C09156=1163.413,-13.561,-45.974,179.721,5.975,149.153
C09157=1163.408,-13.312,-45.986,179.723,5.976,149.152
C09158=1163.403,-13.062,-45.999,179.726,5.976,149.151
C09159=1163.397,-12.812,-46.012,179.728,5.977,149.151
C09160=1163.392,-12.563,-46.025,179.731,5.978,149.150
C09161=1163.388,-12.313,-46.038,179.733,5.978,149.150
C09162=1163.383,-12.063,-46.050,179.736,5.979,149.149
C09163=1163.377,-11.814,-46.064,179.738,5.979,149.148
C09164=1163.372,-11.564,-46.077,179.740,5.980,149.148
C09165=1163.367,-11.314,-46.089,179.743,5.981,149.147
C09166=1163.361,-11.065,-46.102,179.745,5.981,149.147
C09167=1163.356,-10.815,-46.115,179.748,5.982,149.146
C09168=1163.352,-10.565,-46.128,179.750,5.983,149.146
C09169=1163.346,-10.316,-46.141,179.753,5.983,149.145
C09170=1163.341,-10.066,-46.154,179.755,5.984,149.144
C09171=1163.336,-9.816,-46.167,179.758,5.984,149.144
C09172=1163.330,-9.567,-46.180,179.760,5.985,149.143
C09173=1163.326,-9.317,-46.193,179.763,5.986,149.143
C09174=1163.321,-9.067,-46.206,179.766,5.987,149.142
C09175=1163.315,-8.818,-46.219,179.768,5.988,149.141
C09176=1163.311,-8.568,-46.232,179.770,5.988,149.141
C09177=1163.305,-8.319,-46.245,179.773,5.989,149.140
C09178=1163.300,-8.069,-46.258,179.775,5.989,149.140
C09179=1163.295,-7.819,-46.271,179.778,5.990,149.139
C09180=1163.290,-7.570,-46.284,179.780,5.991,149.138
C09181=1163.284,-7.321,-46.297,179.783,5.991,149.138
C09182=1163.280,-7.071,-46.311,179.785,5.992,149.137
C09183=1163.274,-6.822,-46.324,179.788,5.992,149.137
C09184=1163.269,-6.571,-46.337,179.790,5.993,149.136
C09185=1163.264,-6.322,-46.349,179.792,5.994,149.135
C09186=1163.258,-6.073,-46.363,179.795,5.994,149.135
C09187=1163.254,-5.823,-46.376,179.797,5.995,149.134
C09188=1163.248,-5.574,-46.389,179.800,5.995,149.134
C09189=1163.244,-5.323,-46.402,179.802,5.996,149.133
C09190=1163.238,-5.074,-46.416,179.805,5.997,149.132
C09191=1163.233,-4.825,-46.429,179.807,5.997,149.132
C09192=1163.229,-4.575,-46.442,179.810,5.998,149.131
C09193=1163.223,-4.326,-46.455,179.812,5.998,149.131
C09194=1163.218,-4.075,-46.468,179.814,5.999,149.130
C09195=1163.213,-3.826,-46.482,179.817,6.000,149.129
C09196=1163.208,-3.576,-46.495,179.819,6.000,149.129
C09197=1163.202,-3.327,-46.508,179.822,6.002,149.128
C09198=1163.198,-3.077,-46.521,179.825,6.002,149.128
C09199=1163.192,-2.828,-46.535,179.827,6.003,149.127
C09200=1163.187,-2.578,-46.548,179.830,6.003,149.126
C09201=1163.182,-2.328,-46.561,179.832,6.004,149.126
C09202=1163.177,-2.079,-46.575,179.835,6.005,149.125
C09203=1163.172,-1.829,-46.588,179.837,6.006,149.125
C09204=1163.167,-1.580,-46.601,179.840,6.006,149.124
C09205=1163.162,-1.330,-46.615,179.842,6.007,149.124
C09206=1163.157,-1.081,-46.628,179.844,6.007,149.123
C09207=1163.152,-0.831,-46.642,179.847,6.008,149.122
C09208=1163.146,-0.581,-46.655,179.849,6.009,149.122
C09209=1163.141,-0.331,-46.668,179.852,6.009,149.121
C09210=1163.136,-0.082,-46.682,179.854,6.010,149.121
C09211=1163.131,0.168,-46.695,179.857,6.010,149.120
C09212=1163.126,0.417,-46.709,179.860,6.012,149.120
C09213=1163.121,0.667,-46.722,179.862,6.012,149.119
C09214=1163.115,0.916,-46.735,179.865,6.013,149.118
C09215=1163.110,1.166,-46.749,179.867,6.014,149.118
C09216=1163.105,1.415,-46.762,179.870,6.014,149.117
C09217=1163.100,1.685,-46.777,179.872,6.015,149.117
C09218=1163.094,1.954,-46.792,179.874,6.015,149.116
C09219=1163.088,2.223,-46.806,179.878,6.017,149.115
C09220=1163.083,2.493,-46.820,179.880,6.017,149.114
C09221=1163.078,2.742,-46.834,179.883,6.018,149.114
C09222=1163.072,2.992,-46.848,179.885,6.018,149.113
C09223=1163.068,3.241,-46.861,179.887,6.019,149.113
C09224=1163.062,3.491,-46.874,179.890,6.020,149.112
C09225=1163.057,3.741,-46.889,179.893,6.020,149.111
C09226=1163.052,3.990,-46.901,179.895,6.021,149.111
C09227=1163.047,4.240,-46.916,179.898,6.022,149.110
C09228=1163.043,4.490,-46.929,179.900,6.023,149.110
C09229=1163.037,4.739,-46.942,179.903,6.023,149.109
C09230=1163.032,4.988,-46.957,179.905,6.024,149.109
C09231=1163.026,5.238,-46.970,179.908,6.025,149.108
C09232=1163.022,5.487,-46.984,179.910,6.026,149.108
C09233=1163.016,5.737,-46.997,179.913,6.026,149.107
C09234=1163.011,5.987,-47.011,179.915,6.027,149.106
C09235=1163.007,6.236,-47.025,179.917,6.027,149.106
C09236=1163.001,6.486,-47.038,179.921,6.029,149.105
C09237=1162.996,6.736,-47.052,179.923,6.029,149.105
C09238=1162.991,6.985,-47.065,179.925,6.030,149.104
C09239=1162.986,7.235,-47.079,179.928,6.031,149.103
C09240=1162.981,7.484,-47.093,179.930,6.031,149.103
C09241=1162.975,7.734,-47.107,179.933,6.032,149.102
C09242=1162.971,7.983,-47.120,179.935,6.032,149.102
C09243=1162.966,8.233,-47.135,179.938,6.033,149.101
C09244=1162.961,8.482,-47.149,179.941,6.035,149.100
C09245=1162.955,8.732,-47.162,179.943,6.035,149.100
C09246=1162.950,8.981,-47.176,179.945,6.036,149.099
C09247=1162.946,9.231,-47.190,179.948,6.036,149.099
C09248=1162.940,9.481,-47.203,179.950,6.037,149.098
C09249=1162.935,9.730,-47.217,179.953,6.038,149.097
C09250=1162.930,9.980,-47.231,179.955,6.038,149.097
C09251=1162.925,10.229,-47.246,179.958,6.039,149.096
C09252=1162.920,10.479,-47.258,179.961,6.040,149.096
C09253=1162.915,10.729,-47.273,179.963,6.041,149.095
C09254=1162.910,10.978,-47.287,179.966,6.041,149.095
C09255=1162.904,11.227,-47.301,179.968,6.042,149.094
C09256=1162.899,11.478,-47.314,179.971,6.043,149.093
C09257=1162.894,11.727,-47.329,179.973,6.044,149.093
C09258=1162.889,11.976,-47.342,179.975,6.044,149.092
C09259=1162.884,12.226,-47.356,179.979,6.045,149.092
C09260=1162.879,12.475,-47.370,179.981,6.046,149.091
C09261=1162.874,12.724,-47.384,179.983,6.047,149.090
C09262=1162.869,12.975,-47.398,179.986,6.047,149.090
C09263=1162.864,13.224,-47.412,179.988,6.048,149.089
C09264=1162.859,13.474,-47.426,179.990,6.049,149.089
C09265=1162.854,13.723,-47.440,179.993,6.049,149.088
C09266=1162.849,13.973,-47.454,179.996,6.051,149.088
C09267=1162.844,14.222,-47.468,179.998,6.051,149.087
C09268=1162.838,14.471,-47.482,-179.999,6.052,149.086
C09269=1162.833,14.721,-47.497,-179.997,6.053,149.086
C09270=1162.829,14.971,-47.511,-179.994,6.053,149.085
C09271=1162.823,15.221,-47.524,-179.992,6.054,149.085
C09272=1162.818,15.470,-47.538,-179.989,6.055,149.084
C09273=1162.813,15.720,-47.553,-179.986,6.056,149.084
C09274=1162.808,15.969,-47.567,-179.984,6.056,149.083
C09275=1162.803,16.219,-47.581,-179.982,6.057,149.082
C09276=1162.797,16.468,-47.595,-179.979,6.058,149.082
C09277=1162.792,16.718,-47.609,-179.977,6.059,149.081
C09278=1162.787,16.968,-47.624,-179.974,6.060,149.081
C09279=1162.782,17.217,-47.638,-179.971,6.060,149.080
C09280=1162.777,17.466,-47.652,-179.969,6.061,149.079
C09281=1162.772,17.716,-47.666,-179.966,6.062,149.079
C09282=1162.767,17.966,-47.680,-179.964,6.062,149.078
C09283=1162.762,18.215,-47.695,-179.961,6.064,149.078
C09284=1162.757,18.465,-47.709,-179.959,6.065,149.077
C09285=1162.751,18.714,-47.723,-179.956,6.065,149.076
C09286=1162.747,18.964,-47.737,-179.954,6.066,149.076
C09287=1162.742,19.214,-47.751,-179.951,6.066,149.075
C09288=1162.737,19.463,-47.766,-179.948,6.068,149.075
C09289=1162.732,19.712,-47.781,-179.946,6.068,149.074
C09290=1162.726,19.961,-47.795,-179.943,6.069,149.074
C09291=1162.721,20.211,-47.809,-179.941,6.070,149.073
C09292=1162.717,20.461,-47.823,-179.938,6.070,149.072
C09293=1162.712,20.711,-47.837,-179.936,6.071,149.072
C09294=1162.707,20.960,-47.852,-179.933,6.072,149.071
C09295=1162.702,21.210,-47.866,-179.931,6.073,149.071
C09296=1162.696,21.459,-47.880,-179.928,6.074,149.070
C09297=1162.691,21.708,-47.895,-179.926,6.074,149.070
C09298=1162.686,21.958,-47.909,-179.923,6.076,149.069
C09299=1162.682,22.207,-47.923,-179.920,6.077,149.069
C09300=1162.676,22.458,-47.938,-179.918,6.077,149.068
C09301=1162.671,22.707,-47.953,-179.915,6.078,149.067
C09302=1162.666,22.956,-47.968,-179.913,6.078,149.067
C09303=1162.661,23.205,-47.981,-179.910,6.080,149.066
C09304=1162.656,23.455,-47.996,-179.908,6.080,149.066
C09305=1162.651,23.705,-48.010,-179.905,6.081,149.065
C09306=1162.646,23.954,-48.024,-179.903,6.082,149.064
C09307=1162.640,24.204,-48.040,-179.900,6.082,149.064
C09308=1162.635,24.454,-48.054,-179.897,6.084,149.063
C09309=1162.631,24.703,-48.068,-179.895,6.084,149.063
C09310=1162.626,24.953,-48.083,-179.893,6.085,149.062
C09311=1162.621,25.202,-48.098,-179.890,6.086,149.062
C09312=1162.615,25.451,-48.112,-179.887,6.087,149.061
C09313=1162.610,25.701,-48.126,-179.884,6.088,149.060
C09314=1162.605,25.950,-48.141,-179.882,6.088,149.060
C09315=1162.600,26.200,-48.156,-179.880,6.089,149.059
C09316=1162.595,26.450,-48.170,-179.877,6.090,149.059
C09317=1162.590,26.699,-48.185,-179.874,6.091,149.058
C09318=1162.585,26.949,-48.200,-179.872,6.092,149.057
C09319=1162.580,27.198,-48.214,-179.869,6.093,149.057
C09320=1162.575,27.448,-48.229,-179.867,6.093,149.056
C09321=1162.570,27.717,-48.244,-179.864,6.095,149.056
C09322=1162.564,27.986,-48.260,-179.861,6.095,149.055
C09323=1162.559,28.255,-48.276,-179.858,6.096,149.054
C09324=1162.554,28.524,-48.292,-179.856,6.097,149.054
C09325=1162.548,28.772,-48.307,-179.853,6.098,149.053
C09326=1162.543,29.022,-48.321,-179.850,6.099,149.053
C09327=1162.538,29.272,-48.336,-179.848,6.100,149.052
C09328=1162.532,29.521,-48.351,-179.845,6.100,149.052
C09329=1162.527,29.771,-48.365,-179.843,6.101,149.051
C09330=1162.523,30.020,-48.380,-179.840,6.102,149.050
C09331=1162.518,30.270,-48.395,-179.838,6.103,149.050
C09332=1162.512,30.519,-48.410,-179.835,6.104,149.049
C09333=1162.507,30.769,-48.425,-179.833,6.105,149.049
C09334=1162.503,31.018,-48.440,-179.830,6.106,149.048
C09335=1162.497,31.268,-48.454,-179.828,6.107,149.048
C09336=1162.492,31.517,-48.469,-179.825,6.107,149.047
C09337=1162.487,31.767,-48.484,-179.823,6.108,149.047
C09338=1162.482,32.016,-48.499,-179.820,6.109,149.046
C09339=1162.477,32.266,-48.514,-179.817,6.110,149.045
C09340=1162.472,32.515,-48.529,-179.815,6.111,149.045
C09341=1162.467,32.765,-48.543,-179.811,6.112,149.044
C09342=1162.462,33.014,-48.558,-179.809,6.113,149.044
C09343=1162.458,33.264,-48.573,-179.807,6.113,149.043
C09344=1162.452,33.514,-48.589,-179.805,6.114,149.043
C09345=1162.448,33.763,-48.604,-179.801,6.115,149.042
C09346=1162.442,34.013,-48.619,-179.799,6.116,149.041
C09347=1162.437,34.262,-48.634,-179.796,6.117,149.041
C09348=1162.432,34.512,-48.648,-179.794,6.118,149.040
C09349=1162.427,34.761,-48.663,-179.791,6.119,149.040
C09350=1162.422,35.010,-48.678,-179.789,6.120,149.039
C09351=1162.417,35.260,-48.693,-179.786,6.120,149.038
C09352=1162.412,35.509,-48.708,-179.784,6.122,149.038
C09353=1162.407,35.759,-48.724,-179.781,6.122,149.037
C09354=1162.402,36.008,-48.738,-179.779,6.123,149.037
C09355=1162.396,36.258,-48.754,-179.775,6.124,149.036
C09356=1162.392,36.507,-48.769,-179.773,6.125,149.036
C09357=1162.386,36.757,-48.784,-179.771,6.126,149.035
C09358=1162.382,37.007,-48.799,-179.769,6.127,149.035
C09359=1162.377,37.256,-48.814,-179.765,6.128,149.034
C09360=1162.372,37.506,-48.829,-179.763,6.129,149.034
C09361=1162.367,37.755,-48.844,-179.760,6.129,149.033
C09362=1162.362,38.004,-48.859,-179.758,6.131,149.032
C09363=1162.357,38.253,-48.874,-179.755,6.131,149.032
C09364=1162.351,38.503,-48.889,-179.753,6.132,149.031
C09365=1162.346,38.753,-48.905,-179.750,6.134,149.031
C09366=1162.341,39.002,-48.920,-179.748,6.134,149.030
C09367=1162.336,39.252,-48.936,-179.745,6.135,149.030
C09368=1162.331,39.502,-48.950,-179.742,6.137,149.029
C09369=1162.326,39.751,-48.966,-179.739,6.137,149.028
C09370=1162.321,40.000,-48.981,-179.737,6.138,149.028
C09371=1162.316,40.250,-48.996,-179.735,6.138,149.027
C09372=1162.311,40.499,-49.011,-179.732,6.140,149.027
C09373=1162.306,40.748,-49.027,-179.729,6.140,149.026
C09374=1162.301,40.999,-49.042,-179.727,6.141,149.026
C09375=1162.296,41.248,-49.057,-179.724,6.143,149.025
C09376=1162.291,41.497,-49.073,-179.722,6.143,149.025
C09377=1162.286,41.746,-49.088,-179.719,6.144,149.024
C09378=1162.281,41.996,-49.103,-179.716,6.146,149.023
C09379=1162.277,42.246,-49.119,-179.714,6.146,149.023
C09380=1162.271,42.495,-49.134,-179.712,6.147,149.022
C09381=1162.266,42.744,-49.150,-179.708,6.148,149.022
C09382=1162.261,42.994,-49.165,-179.706,6.149,149.021
C09383=1162.256,43.244,-49.180,-179.704,6.150,149.021
C09384=1162.251,43.494,-49.196,-179.701,6.151,149.020
C09385=1162.246,43.743,-49.211,-179.698,6.152,149.019
C09386=1162.241,43.992,-49.226,-179.696,6.153,149.019
C09387=1162.235,44.242,-49.242,-179.693,6.154,149.018
C09388=1162.231,44.491,-49.257,-179.691,6.155,149.018
C09389=1162.226,44.741,-49.273,-179.687,6.156,149.017
C09390=1162.221,44.990,-49.288,-179.685,6.157,149.017
C09391=1162.216,45.239,-49.303,-179.683,6.157,149.016
C09392=1162.211,45.489,-49.319,-179.680,6.159,149.016
C09393=1162.206,45.739,-49.335,-179.677,6.160,149.015
C09394=1162.201,45.988,-49.350,-179.675,6.160,149.015
C09395=1162.196,46.237,-49.365,-179.672,6.162,149.014
C09396=1162.190,46.487,-49.381,-179.670,6.163,149.013
C09397=1162.186,46.737,-49.397,-179.667,6.163,149.013
C09398=1162.181,46.985,-49.413,-179.664,6.165,149.012
C09399=1162.176,47.235,-49.428,-179.662,6.165,149.012
C09400=1162.171,47.484,-49.444,-179.659,6.166,149.011
C09401=1162.166,47.734,-49.459,-179.656,6.167,149.011
C09402=1162.161,47.983,-49.475,-179.654,6.168,149.010
C09403=1162.156,48.233,-49.490,-179.651,6.169,149.009
C09404=1162.151,48.483,-49.506,-179.649,6.170,149.009
C09405=1162.146,48.732,-49.522,-179.646,6.171,149.008
C09406=1162.141,48.981,-49.537,-179.643,6.172,149.008
C09407=1162.136,49.231,-49.554,-179.641,6.173,149.007
C09408=1162.131,49.480,-49.569,-179.638,6.174,149.007
C09409=1162.126,49.730,-49.585,-179.635,6.175,149.006
C09410=1162.121,49.979,-49.600,-179.633,6.176,149.006
C09411=1162.116,50.229,-49.616,-179.630,6.178,149.005
C09412=1162.111,50.478,-49.632,-179.628,6.178,149.005
C09413=1162.106,50.727,-49.648,-179.626,6.179,149.004
C09414=1162.101,50.977,-49.664,-179.622,6.180,149.003
C09415=1162.096,51.226,-49.679,-179.620,6.181,149.003
C09416=1162.091,51.476,-49.694,-179.617,6.182,149.002
C09417=1162.086,51.725,-49.711,-179.615,6.183,149.002
C09418=1162.081,51.974,-49.726,-179.612,6.184,149.001
C09419=1162.076,52.225,-49.742,-179.609,6.185,149.001
C09420=1162.071,52.474,-49.758,-179.607,6.186,149.000
C09421=1162.066,52.723,-49.774,-179.604,6.188,149.000
C09422=1162.061,52.973,-49.790,-179.601,6.188,148.999
C09423=1162.056,53.222,-49.806,-179.599,6.189,148.999
C09424=1162.051,53.471,-49.821,-179.596,6.190,148.998
C09425=1162.046,53.740,-49.839,-179.594,6.191,148.997
C09426=1162.041,54.008,-49.856,-179.591,6.192,148.997
C09427=1162.035,54.277,-49.873,-179.587,6.194,148.996
C09428=1162.030,54.545,-49.890,-179.585,6.195,148.996
C09429=1162.025,54.795,-49.906,-179.582,6.196,148.995
C09430=1162.020,55.044,-49.922,-179.580,6.197,148.995
C09431=1162.015,55.294,-49.938,-179.577,6.197,148.994
C09432=1162.010,55.544,-49.954,-179.574,6.199,148.993
C09433=1162.005,55.792,-49.970,-179.572,6.199,148.993
C09434=1162.000,56.043,-49.986,-179.569,6.201,148.992
C09435=1161.995,56.291,-50.002,-179.567,6.202,148.992
C09436=1161.990,56.541,-50.018,-179.564,6.203,148.991
C09437=1161.985,56.790,-50.035,-179.562,6.204,148.991
C09438=1161.980,57.040,-50.050,-179.559,6.205,148.990
C09439=1161.975,57.290,-50.066,-179.556,6.206,148.990
C09440=1161.970,57.539,-50.082,-179.554,6.207,148.989
C09441=1161.965,57.789,-50.098,-179.551,6.208,148.989
C09442=1161.960,58.037,-50.115,-179.548,6.209,148.988
C09443=1161.955,58.288,-50.131,-179.545,6.211,148.988
C09444=1161.950,58.536,-50.147,-179.543,6.211,148.987
C09445=1161.945,58.786,-50.163,-179.541,6.212,148.986
C09446=1161.940,59.035,-50.179,-179.538,6.214,148.986
C09447=1161.935,59.285,-50.195,-179.535,6.214,148.985
C09448=1161.930,59.534,-50.211,-179.533,6.216,148.985
C09449=1161.926,59.784,-50.228,-179.530,6.216,148.984
C09450=1161.920,60.033,-50.244,-179.527,6.218,148.984
C09451=1161.915,60.283,-50.261,-179.525,6.219,148.983
C09452=1161.910,60.532,-50.277,-179.522,6.220,148.983
C09453=1161.905,60.782,-50.293,-179.519,6.221,148.982
C09454=1161.900,61.031,-50.309,-179.517,6.222,148.982
C09455=1161.895,61.281,-50.325,-179.514,6.223,148.981
C09456=1161.890,61.529,-50.342,-179.512,6.224,148.980
C09457=1161.885,61.779,-50.358,-179.509,6.225,148.980
C09458=1161.880,62.028,-50.374,-179.506,6.226,148.979
C09459=1161.876,62.278,-50.391,-179.503,6.228,148.979
C09460=1161.870,62.527,-50.407,-179.501,6.228,148.978
C09461=1161.865,62.777,-50.424,-179.498,6.230,148.978
C09462=1161.860,63.026,-50.440,-179.496,6.231,148.977
C09463=1161.855,63.276,-50.456,-179.493,6.232,148.977
C09464=1161.851,63.525,-50.472,-179.491,6.233,148.976
C09465=1161.846,63.774,-50.489,-179.487,6.234,148.976
C09466=1161.840,64.024,-50.505,-179.485,6.235,148.975
C09467=1161.835,64.273,-50.522,-179.482,6.236,148.975
C09468=1161.831,64.523,-50.538,-179.480,6.237,148.974
C09469=1161.826,64.772,-50.555,-179.477,6.238,148.973
C09470=1161.821,65.022,-50.571,-179.474,6.239,148.973
C09471=1161.816,65.271,-50.587,-179.472,6.240,148.973
C09472=1161.811,65.520,-50.604,-179.469,6.242,148.972
C09473=1161.806,65.770,-50.621,-179.467,6.242,148.971
C09474=1161.801,66.019,-50.636,-179.464,6.244,148.971
C09475=1161.796,66.269,-50.653,-179.462,6.245,148.970
C09476=1161.791,66.518,-50.670,-179.459,6.246,148.970
C09477=1161.786,66.767,-50.687,-179.456,6.247,148.969
C09478=1161.781,67.017,-50.703,-179.453,6.248,148.969
C09479=1161.776,67.265,-50.720,-179.451,6.249,148.968
C09480=1161.771,67.516,-50.736,-179.448,6.251,148.968
C09481=1161.766,67.765,-50.753,-179.445,6.251,148.967
C09482=1161.761,68.014,-50.769,-179.443,6.253,148.967
C09483=1161.757,68.264,-50.786,-179.441,6.254,148.966
C09484=1161.752,68.513,-50.803,-179.437,6.255,148.966
C09485=1161.746,68.762,-50.819,-179.435,6.256,148.965
C09486=1161.742,69.012,-50.836,-179.432,6.257,148.964
C09487=1161.737,69.261,-50.853,-179.430,6.258,148.964
C09488=1161.732,69.510,-50.870,-179.427,6.260,148.964
C09489=1161.727,69.760,-50.886,-179.424,6.260,148.963
C09490=1161.722,70.010,-50.903,-179.422,6.262,148.963
C09491=1161.717,70.259,-50.919,-179.419,6.262,148.962
C09492=1161.712,70.508,-50.936,-179.416,6.264,148.961
C09493=1161.707,70.758,-50.953,-179.413,6.265,148.961
C09494=1161.702,71.007,-50.969,-179.411,6.266,148.960
C09495=1161.697,71.257,-50.987,-179.408,6.268,148.960
C09496=1161.692,71.506,-51.003,-179.406,6.268,148.959
C09497=1161.687,71.755,-51.020,-179.403,6.270,148.959
C09498=1161.682,72.005,-51.037,-179.400,6.271,148.958
C09499=1161.677,72.254,-51.053,-179.398,6.272,148.958
C09500=1161.673,72.504,-51.070,-179.395,6.273,148.957
C09501=1161.667,72.753,-51.087,-179.392,6.275,148.957
C09502=1161.663,73.002,-51.104,-179.390,6.275,148.956
C09503=1161.658,73.252,-51.122,-179.387,6.277,148.956
C09504=1161.653,73.500,-51.138,-179.385,6.278,148.955
C09505=1161.647,73.750,-51.155,-179.382,6.279,148.955
C09506=1161.643,74.000,-51.172,-179.379,6.280,148.954
C09507=1161.638,74.249,-51.189,-179.377,6.281,148.954
C09508=1161.633,74.498,-51.206,-179.373,6.283,148.953
C09509=1161.628,74.748,-51.222,-179.371,6.284,148.953
C09510=1161.623,74.997,-51.239,-179.368,6.285,148.952
C09511=1161.619,75.246,-51.257,-179.366,6.286,148.951
C09512=1161.613,75.495,-51.274,-179.363,6.288,148.951
C09513=1161.608,75.745,-51.290,-179.361,6.288,148.951
C09514=1161.603,75.995,-51.308,-179.358,6.290,148.950
C09515=1161.599,76.244,-51.324,-179.356,6.291,148.950
C09516=1161.593,76.494,-51.342,-179.352,6.292,148.949
C09517=1161.589,76.742,-51.359,-179.350,6.294,148.948
C09518=1161.583,76.992,-51.376,-179.347,6.294,148.948
C09519=1161.579,77.241,-51.393,-179.344,6.296,148.947
C09520=1161.574,77.491,-51.410,-179.342,6.297,148.947
C09521=1161.569,77.740,-51.428,-179.339,6.298,148.946
C09522=1161.564,77.989,-51.444,-179.337,6.299,148.946
C09523=1161.559,78.239,-51.461,-179.334,6.301,148.945
C09524=1161.554,78.488,-51.478,-179.331,6.301,148.945
C09525=1161.549,78.738,-51.496,-179.329,6.303,148.944
C09526=1161.545,78.987,-51.513,-179.326,6.304,148.944
C09527=1161.539,79.237,-51.530,-179.323,6.305,148.943
C09528=1161.534,79.485,-51.548,-179.321,6.307,148.943
C09529=1161.529,79.754,-51.566,-179.317,6.308,148.942
C09530=1161.524,80.023,-51.584,-179.315,6.309,148.942
C09531=1161.518,80.291,-51.603,-179.312,6.310,148.941
C09532=1161.514,80.559,-51.621,-179.309,6.312,148.941
C09533=1161.508,80.809,-51.639,-179.306,6.313,148.940
C09534=1161.503,81.059,-51.656,-179.304,6.314,148.940
C09535=1161.499,81.307,-51.673,-179.301,6.316,148.939
C09536=1161.493,81.556,-51.690,-179.299,6.316,148.939
C09537=1161.488,81.806,-51.708,-179.296,6.318,148.938
C09538=1161.484,82.055,-51.725,-179.293,6.318,148.937
C09539=1161.479,82.305,-51.742,-179.290,6.320,148.937
C09540=1161.474,82.554,-51.760,-179.288,6.322,148.937
C09541=1161.469,82.804,-51.777,-179.285,6.322,148.936
C09542=1161.464,83.053,-51.795,-179.282,6.324,148.936
C09543=1161.459,83.303,-51.812,-179.280,6.325,148.935
C09544=1161.455,83.551,-51.829,-179.277,6.326,148.934
C09545=1161.450,83.801,-51.847,-179.274,6.328,148.934
C09546=1161.444,84.050,-51.864,-179.272,6.329,148.934
C09547=1161.439,84.299,-51.882,-179.269,6.330,148.933
C09548=1161.435,84.548,-51.899,-179.266,6.332,148.933
C09549=1161.430,84.798,-51.916,-179.264,6.333,148.932
C09550=1161.425,85.047,-51.934,-179.261,6.334,148.931
C09551=1161.419,85.297,-51.952,-179.259,6.335,148.931
C09552=1161.415,85.546,-51.969,-179.256,6.337,148.931
C09553=1161.410,85.796,-51.986,-179.253,6.338,148.930
C09554=1161.405,86.045,-52.004,-179.251,6.339,148.930
C09555=1161.400,86.294,-52.022,-179.247,6.340,148.929
C09556=1161.395,86.544,-52.039,-179.245,6.342,148.928
C09557=1161.391,86.793,-52.057,-179.243,6.343,148.928
C09558=1161.386,87.043,-52.074,-179.239,6.344,148.927
C09559=1161.381,87.292,-52.092,-179.237,6.345,148.927
C09560=1161.376,87.541,-52.110,-179.234,6.347,148.927
C09561=1161.371,87.791,-52.127,-179.231,6.348,148.926
C09562=1161.366,88.040,-52.145,-179.229,6.349,148.925
C09563=1161.361,88.289,-52.163,-179.226,6.351,148.925
C09564=1161.356,88.539,-52.180,-179.223,6.352,148.924
C09565=1161.351,88.788,-52.198,-179.221,6.353,148.924
C09566=1161.346,89.037,-52.216,-179.218,6.354,148.924
C09567=1161.341,89.287,-52.233,-179.215,6.356,148.923
C09568=1161.336,89.536,-52.251,-179.213,6.357,148.922
C09569=1161.332,89.785,-52.268,-179.210,6.358,148.922
C09570=1161.327,90.034,-52.286,-179.208,6.359,148.922
C09571=1161.322,90.284,-52.304,-179.205,6.361,148.921
C09572=1161.317,90.533,-52.322,-179.202,6.362,148.921
C09573=1161.312,90.782,-52.340,-179.200,6.363,148.920
C09574=1161.307,91.031,-52.358,-179.197,6.364,148.920
C09575=1161.302,91.280,-52.376,-179.194,6.366,148.919
C09576=1161.297,91.530,-52.393,-179.192,6.367,148.919
C09577=1161.292,91.779,-52.411,-179.189,6.368,148.918
C09578=1161.287,92.029,-52.429,-179.186,6.370,148.918
C09579=1161.282,92.278,-52.447,-179.184,6.371,148.917
C09580=1161.278,92.528,-52.465,-179.181,6.372,148.917
C09581=1161.273,92.777,-52.483,-179.178,6.374,148.916
C09582=1161.268,93.027,-52.500,-179.176,6.375,148.916
C09583=1161.263,93.276,-52.518,-179.173,6.376,148.915
C09584=1161.258,93.525,-52.536,-179.170,6.378,148.915
C09585=1161.253,93.774,-52.554,-179.168,6.379,148.914
C09586=1161.248,94.023,-52.572,-179.164,6.380,148.914
C09587=1161.243,94.272,-52.590,-179.162,6.382,148.913
C09588=1161.238,94.522,-52.608,-179.159,6.384,148.913
C09589=1161.234,94.771,-52.626,-179.157,6.384,148.912
C09590=1161.229,95.021,-52.645,-179.154,6.386,148.912
C09591=1161.224,95.270,-52.663,-179.151,6.387,148.911
C09592=1161.219,95.519,-52.681,-179.149,6.388,148.911
C09593=1161.214,95.768,-52.699,-179.146,6.390,148.910
C09594=1161.210,96.017,-52.717,-179.143,6.391,148.910
C09595=1161.205,96.267,-52.735,-179.141,6.392,148.909
C09596=1161.200,96.516,-52.753,-179.137,6.394,148.909
C09597=1161.195,96.765,-52.771,-179.135,6.395,148.908
C09598=1161.191,97.015,-52.789,-179.133,6.396,148.908
C09599=1161.186,97.264,-52.807,-179.130,6.398,148.907
C09600=1161.181,97.513,-52.825,-179.127,6.399,148.907
C09601=1161.176,97.762,-52.843,-179.124,6.401,148.906
C09602=1161.170,98.012,-52.861,-179.122,6.402,148.906
C09603=1161.166,98.262,-52.880,-179.119,6.403,148.905
C09604=1161.161,98.511,-52.898,-179.116,6.405,148.905
C09605=1161.156,98.760,-52.916,-179.114,6.406,148.905
C09606=1161.151,99.009,-52.934,-179.111,6.407,148.904
C09607=1161.146,99.258,-52.952,-179.108,6.409,148.903
C09608=1161.141,99.508,-52.970,-179.105,6.410,148.903
C09609=1161.137,99.757,-52.989,-179.103,6.411,148.903
C09610=1161.132,100.006,-53.007,-179.100,6.413,148.902
C09611=1161.127,100.256,-53.025,-179.097,6.414,148.902
C09612=1161.122,100.505,-53.043,-179.095,6.415,148.901
C09613=1161.117,100.755,-53.062,-179.092,6.417,148.901
C09614=1161.113,101.004,-53.080,-179.089,6.418,148.900
C09615=1161.107,101.253,-53.099,-179.086,6.420,148.900
C09616=1161.102,101.502,-53.117,-179.084,6.421,148.899
C09617=1161.098,101.752,-53.135,-179.081,6.423,148.899
C09618=1161.093,102.001,-53.153,-179.078,6.424,148.898
C09619=1161.088,102.250,-53.172,-179.075,6.426,148.898
C09620=1161.083,102.499,-53.190,-179.073,6.427,148.897
C09621=1161.079,102.749,-53.209,-179.071,6.428,148.897
C09622=1161.074,102.998,-53.227,-179.067,6.430,148.896
C09623=1161.068,103.247,-53.246,-179.065,6.431,148.896
C09624=1161.063,103.496,-53.264,-179.063,6.432,148.896
C09625=1161.059,103.746,-53.282,-179.060,6.434,148.895
C09626=1161.054,103.994,-53.301,-179.057,6.435,148.895
C09627=1161.049,104.244,-53.320,-179.054,6.437,148.894
C09628=1161.044,104.494,-53.338,-179.052,6.438,148.894
C09629=1161.040,104.742,-53.357,-179.049,6.439,148.893
C09630=1161.034,104.992,-53.375,-179.046,6.441,148.893
C09631=1161.029,105.241,-53.393,-179.043,6.443,148.892
C09632=1161.025,105.490,-53.412,-179.041,6.444,148.892
C09633=1161.019,105.759,-53.432,-179.038,6.445,148.891
C09634=1161.014,106.027,-53.452,-179.035,6.447,148.891
C09635=1161.009,106.295,-53.472,-179.032,6.448,148.890
C09636=1161.004,106.564,-53.492,-179.029,6.450,148.890
C09637=1160.999,106.813,-53.511,-179.026,6.451,148.889
C09638=1160.994,107.062,-53.529,-179.024,6.453,148.889
C09639=1160.990,107.312,-53.548,-179.020,6.454,148.888
C09640=1160.984,107.561,-53.567,-179.018,6.455,148.888
C09641=1160.980,107.810,-53.585,-179.016,6.457,148.887
C09642=1160.975,108.059,-53.605,-179.013,6.459,148.887
C09643=1160.970,108.309,-53.623,-179.010,6.460,148.886
C09644=1160.966,108.558,-53.642,-179.008,6.461,148.886
C09645=1160.960,108.807,-53.660,-179.005,6.463,148.886
C09646=1160.956,109.056,-53.679,-179.002,6.464,148.885
C09647=1160.951,109.306,-53.698,-178.999,6.466,148.885
C09648=1160.946,109.555,-53.717,-178.996,6.467,148.884
C09649=1160.940,109.804,-53.735,-178.994,6.468,148.884
C09650=1160.936,110.053,-53.754,-178.991,6.470,148.883
C09651=1160.931,110.302,-53.774,-178.989,6.472,148.883
C09652=1160.927,110.552,-53.792,-178.985,6.473,148.882
C09653=1160.921,110.801,-53.811,-178.983,6.475,148.882
C09654=1160.917,111.051,-53.830,-178.981,6.476,148.881
C09655=1160.912,111.299,-53.848,-178.978,6.477,148.881
C09656=1160.907,111.548,-53.868,-178.975,6.479,148.881
C09657=1160.902,111.799,-53.887,-178.972,6.480,148.880
C09658=1160.897,112.047,-53.905,-178.969,6.482,148.880
C09659=1160.893,112.297,-53.925,-178.967,6.483,148.879
C09660=1160.888,112.546,-53.943,-178.964,6.485,148.879
C09661=1160.883,112.795,-53.962,-178.961,6.486,148.878
C09662=1160.878,113.044,-53.981,-178.958,6.488,148.878
C09663=1160.873,113.293,-54.000,-178.956,6.490,148.877
C09664=1160.869,113.543,-54.019,-178.954,6.490,148.877
C09665=1160.863,113.792,-54.038,-178.951,6.492,148.877
C09666=1160.859,114.041,-54.056,-178.948,6.493,148.876
C09667=1160.854,114.290,-54.076,-178.945,6.495,148.875
C09668=1160.849,114.540,-54.095,-178.942,6.497,148.875
C09669=1160.844,114.788,-54.114,-178.940,6.499,148.875
C09670=1160.840,115.038,-54.134,-178.937,6.500,148.874
C09671=1160.834,115.288,-54.152,-178.934,6.501,148.874
C09672=1160.830,115.537,-54.171,-178.932,6.503,148.873
C09673=1160.825,115.786,-54.191,-178.929,6.504,148.873
C09674=1160.821,116.035,-54.210,-178.926,6.506,148.872
C09675=1160.815,116.284,-54.229,-178.923,6.508,148.872
C09676=1160.810,116.534,-54.248,-178.921,6.509,148.872
C09677=1160.806,116.782,-54.267,-178.918,6.510,148.871
C09678=1160.801,117.032,-54.286,-178.915,6.512,148.871
C09679=1160.796,117.281,-54.306,-178.913,6.513,148.870
C09680=1160.792,117.530,-54.325,-178.910,6.515,148.870
C09681=1160.786,117.779,-54.344,-178.907,6.517,148.869
C09682=1160.782,118.029,-54.364,-178.905,6.517,148.869
C09683=1160.778,118.278,-54.383,-178.902,6.519,148.868
C09684=1160.772,118.527,-54.402,-178.899,6.521,148.868
C09685=1160.767,118.776,-54.422,-178.896,6.523,148.868
C09686=1160.762,119.026,-54.440,-178.894,6.524,148.867
C09687=1160.758,119.275,-54.459,-178.891,6.526,148.867
C09688=1160.752,119.524,-54.479,-178.888,6.527,148.866
C09689=1160.748,119.774,-54.498,-178.886,6.528,148.866
C09690=1160.743,120.023,-54.518,-178.883,6.530,148.865
C09691=1160.738,120.272,-54.537,-178.880,6.532,148.865
C09692=1160.734,120.521,-54.556,-178.878,6.533,148.865
C09693=1160.728,120.770,-54.576,-178.875,6.535,148.864
C09694=1160.723,121.020,-54.595,-178.872,6.536,148.863
C09695=1160.720,121.268,-54.615,-178.869,6.538,148.863
C09696=1160.714,121.517,-54.634,-178.866,6.540,148.863
C09697=1160.710,121.767,-54.654,-178.864,6.541,148.862
C09698=1160.704,122.016,-54.673,-178.861,6.542,148.862
C09699=1160.700,122.265,-54.693,-178.859,6.544,148.861
C09700=1160.696,122.514,-54.712,-178.856,6.546,148.861
C09701=1160.690,122.763,-54.731,-178.853,6.547,148.860
C09702=1160.686,123.013,-54.751,-178.850,6.549,148.860
C09703=1160.681,123.262,-54.771,-178.847,6.551,148.860
C09704=1160.675,123.511,-54.790,-178.845,6.552,148.859
C09705=1160.671,123.760,-54.810,-178.842,6.553,148.859
C09706=1160.667,124.009,-54.829,-178.840,6.555,148.858
C09707=1160.662,124.258,-54.849,-178.837,6.557,148.858
C09708=1160.657,124.508,-54.868,-178.834,6.558,148.857
C09709=1160.652,124.757,-54.888,-178.831,6.560,148.857
C09710=1160.647,125.006,-54.908,-178.828,6.562,148.857
C09711=1160.642,125.255,-54.927,-178.826,6.563,148.856
C09712=1160.638,125.505,-54.947,-178.823,6.565,148.856
C09713=1160.632,125.754,-54.966,-178.820,6.567,148.855
C09714=1160.628,126.003,-54.986,-178.818,6.568,148.855
C09715=1160.623,126.252,-55.006,-178.815,6.569,148.854
C09716=1160.619,126.502,-55.026,-178.812,6.571,148.854
C09717=1160.614,126.750,-55.045,-178.810,6.572,148.854
C09718=1160.609,126.999,-55.065,-178.807,6.574,148.853
C09719=1160.605,127.249,-55.085,-178.804,6.576,148.853
C09720=1160.599,127.498,-55.104,-178.801,6.578,148.852
C09721=1160.595,127.747,-55.125,-178.799,6.579,148.852
C09722=1160.590,127.996,-55.144,-178.796,6.581,148.852
C09723=1160.585,128.246,-55.164,-178.793,6.582,148.851
C09724=1160.580,128.494,-55.184,-178.790,6.584,148.851
C09725=1160.576,128.744,-55.203,-178.787,6.586,148.850
C09726=1160.571,128.993,-55.223,-178.785,6.588,148.850
C09727=1160.566,129.242,-55.244,-178.782,6.589,148.849
C09728=1160.561,129.491,-55.263,-178.780,6.590,148.849
C09729=1160.557,129.740,-55.283,-178.777,6.592,148.849
C09730=1160.552,129.990,-55.303,-178.774,6.594,148.848
C09731=1160.547,130.239,-55.322,-178.772,6.595,148.848
C09732=1160.542,130.488,-55.343,-178.769,6.597,148.847
C09733=1160.537,130.737,-55.363,-178.766,6.598,148.847
C09734=1160.532,130.986,-55.383,-178.763,6.600,148.846
C09735=1160.527,131.236,-55.403,-178.760,6.602,148.846
C09736=1160.523,131.485,-55.423,-178.758,6.604,148.846
C09737=1160.518,131.753,-55.444,-178.755,6.605,148.845
C09738=1160.512,132.022,-55.466,-178.752,6.607,148.845
C09739=1160.508,132.290,-55.488,-178.748,6.609,148.844
C09740=1160.502,132.559,-55.509,-178.746,6.611,148.844
C09741=1160.497,132.808,-55.529,-178.743,6.613,148.843
C09742=1160.492,133.057,-55.549,-178.740,6.614,148.843
C09743=1160.488,133.306,-55.569,-178.738,6.616,148.843
C09744=1160.483,133.556,-55.589,-178.735,6.618,148.842
C09745=1160.479,133.805,-55.609,-178.733,6.619,148.842
C09746=1160.474,134.054,-55.630,-178.730,6.620,148.842
C09747=1160.469,134.303,-55.650,-178.727,6.622,148.841
C09748=1160.464,134.552,-55.670,-178.724,6.624,148.841
C09749=1160.459,134.801,-55.690,-178.721,6.625,148.840
C09750=1160.455,135.050,-55.710,-178.719,6.627,148.840
C09751=1160.449,135.299,-55.731,-178.716,6.629,148.839
C09752=1160.445,135.549,-55.751,-178.713,6.630,148.839
C09753=1160.440,135.798,-55.771,-178.711,6.632,148.839
C09754=1160.436,136.047,-55.791,-178.708,6.634,148.838
C09755=1160.431,136.296,-55.811,-178.705,6.636,148.838
C09756=1160.425,136.545,-55.832,-178.703,6.637,148.837
C09757=1160.421,136.794,-55.852,-178.700,6.639,148.837
C09758=1160.416,137.043,-55.872,-178.697,6.641,148.837
C09759=1160.412,137.293,-55.892,-178.694,6.643,148.836
C09760=1160.406,137.542,-55.913,-178.692,6.644,148.836
C09761=1160.402,137.791,-55.933,-178.689,6.646,148.835
C09762=1160.398,138.040,-55.954,-178.686,6.648,148.835
C09763=1160.392,138.289,-55.975,-178.684,6.649,148.835
C09764=1160.388,138.539,-55.994,-178.680,6.651,148.834
C09765=1160.383,138.787,-56.015,-178.678,6.653,148.834
C09766=1160.379,139.036,-56.035,-178.675,6.654,148.833
C09767=1160.374,139.286,-56.056,-178.672,6.656,148.833
C09768=1160.369,139.535,-56.077,-178.670,6.658,148.832
C09769=1160.365,139.784,-56.097,-178.667,6.659,148.832
C09770=1160.359,140.033,-56.117,-178.664,6.661,148.832
C09771=1160.355,140.282,-56.138,-178.661,6.663,148.831
C09772=1160.350,140.531,-56.158,-178.659,6.665,148.831
C09773=1160.345,140.781,-56.179,-178.656,6.666,148.831
C09774=1160.341,141.030,-56.199,-178.653,6.668,148.830
C09775=1160.336,141.279,-56.220,-178.651,6.670,148.830
C09776=1160.331,141.528,-56.241,-178.648,6.672,148.829
C09777=1160.327,141.777,-56.261,-178.645,6.673,148.829
C09778=1160.322,142.026,-56.282,-178.643,6.675,148.829
C09779=1160.317,142.275,-56.302,-178.640,6.677,148.828
C09780=1160.312,142.524,-56.323,-178.637,6.678,148.828
C09781=1160.308,142.773,-56.344,-178.634,6.680,148.827
C09782=1160.303,143.022,-56.364,-178.632,6.682,148.827
C09783=1160.298,143.271,-56.385,-178.629,6.684,148.827
C09784=1160.293,143.520,-56.405,-178.626,6.685,148.826
C09785=1160.288,143.770,-56.426,-178.623,6.688,148.826
C09786=1160.284,144.018,-56.447,-178.620,6.690,148.826
C09787=1160.279,144.268,-56.468,-178.618,6.691,148.825
C09788=1160.274,144.517,-56.488,-178.615,6.693,148.825
C09789=1160.269,144.766,-56.509,-178.612,6.695,148.824
C09790=1160.265,145.015,-56.529,-178.609,6.697,148.824
C09791=1160.259,145.264,-56.550,-178.607,6.698,148.824
C09792=1160.255,145.513,-56.571,-178.604,6.700,148.823
C09793=1160.250,145.762,-56.592,-178.601,6.702,148.823
C09794=1160.246,146.011,-56.613,-178.599,6.704,148.822
C09795=1160.241,146.261,-56.634,-178.596,6.705,148.822
C09796=1160.237,146.510,-56.654,-178.593,6.707,148.822
C09797=1160.232,146.759,-56.675,-178.591,6.709,148.821
C09798=1160.227,147.008,-56.696,-178.588,6.710,148.821
C09799=1160.222,147.257,-56.717,-178.585,6.712,148.821
C09800=1160.217,147.506,-56.738,-178.582,6.714,148.820
C09801=1160.213,147.755,-56.759,-178.580,6.716,148.820
C09802=1160.207,148.004,-56.780,-178.577,6.717,148.819
C09803=1160.203,148.253,-56.800,-178.574,6.719,148.819
C09804=1160.199,148.502,-56.822,-178.571,6.722,148.819
C09805=1160.194,148.751,-56.843,-178.568,6.723,148.818
C09806=1160.189,149.000,-56.864,-178.566,6.725,148.818
C09807=1160.184,149.250,-56.885,-178.563,6.727,148.818
C09808=1160.180,149.498,-56.906,-178.560,6.729,148.817
C09809=1160.175,149.747,-56.927,-178.558,6.730,148.817
C09810=1160.169,149.997,-56.948,-178.555,6.732,148.816
C09811=1160.166,150.246,-56.969,-178.552,6.734,148.816
C09812=1160.161,150.495,-56.990,-178.549,6.736,148.816
C09813=1160.156,150.744,-57.011,-178.547,6.737,148.815
C09814=1160.151,150.992,-57.032,-178.544,6.739,148.815
C09815=1160.146,151.242,-57.053,-178.541,6.741,148.814
C09816=1160.141,151.491,-57.074,-178.538,6.743,148.814
C09817=1160.138,151.740,-57.095,-178.535,6.745,148.814
C09818=1160.132,151.989,-57.116,-178.533,6.747,148.813
C09819=1160.128,152.238,-57.138,-178.530,6.749,148.813
C09820=1160.122,152.487,-57.159,-178.527,6.750,148.813
C09821=1160.119,152.736,-57.180,-178.525,6.752,148.812
C09822=1160.114,152.985,-57.201,-178.522,6.754,148.812
C09823=1160.108,153.235,-57.222,-178.520,6.756,148.812
C09824=1160.104,153.483,-57.244,-178.517,6.758,148.811
C09825=1160.099,153.732,-57.264,-178.514,6.759,148.811
C09826=1160.095,153.982,-57.287,-178.511,6.762,148.811
C09827=1160.090,154.231,-57.307,-178.508,6.764,148.810
C09828=1160.085,154.479,-57.329,-178.506,6.765,148.810
C09829=1160.080,154.729,-57.350,-178.503,6.767,148.809
C09830=1160.076,154.978,-57.372,-178.500,6.769,148.809
C09831=1160.071,155.226,-57.393,-178.497,6.771,148.809
C09832=1160.066,155.476,-57.414,-178.495,6.772,148.808
C09833=1160.061,155.724,-57.436,-178.492,6.774,148.808
C09834=1160.057,155.974,-57.457,-178.489,6.777,148.808
C09835=1160.053,156.223,-57.478,-178.486,6.778,148.807
C09836=1160.047,156.472,-57.499,-178.483,6.780,148.807
C09837=1160.043,156.721,-57.521,-178.481,6.782,148.807
C09838=1160.038,156.970,-57.543,-178.478,6.784,148.806
C09839=1160.033,157.219,-57.564,-178.476,6.786,148.806
C09840=1160.029,157.468,-57.586,-178.473,6.787,148.805
C09841=1160.023,157.737,-57.608,-178.470,6.790,148.805
C09842=1160.018,158.006,-57.633,-178.467,6.792,148.805
C09843=1160.014,158.275,-57.655,-178.464,6.793,148.804
C09844=1160.008,158.544,-57.679,-178.461,6.796,148.804
C09845=1160.004,158.793,-57.701,-178.458,6.798,148.804
C09846=1159.999,159.042,-57.722,-178.456,6.799,148.803
C09847=1159.994,159.291,-57.743,-178.453,6.801,148.803
C09848=1159.990,159.540,-57.765,-178.450,6.803,148.803
C09849=1159.985,159.789,-57.786,-178.447,6.805,148.802
C09850=1159.980,160.037,-57.808,-178.444,6.807,148.802
C09851=1159.976,160.287,-57.829,-178.442,6.809,148.801
C09852=1159.971,160.536,-57.851,-178.439,6.811,148.801
C09853=1159.966,160.785,-57.873,-178.436,6.812,148.801
C09854=1159.962,161.034,-57.895,-178.434,6.814,148.801
C09855=1159.957,161.283,-57.917,-178.431,6.817,148.800
C09856=1159.953,161.532,-57.939,-178.428,6.819,148.800
C09857=1159.948,161.781,-57.960,-178.425,6.821,148.799
C09858=1159.943,162.030,-57.981,-178.423,6.822,148.799
C09859=1159.938,162.279,-58.003,-178.420,6.824,148.799
C09860=1159.934,162.528,-58.025,-178.417,6.826,148.798
C09861=1159.929,162.777,-58.047,-178.414,6.828,148.798
C09862=1159.924,163.026,-58.069,-178.412,6.830,148.798
C09863=1159.920,163.275,-58.090,-178.409,6.832,148.797
C09864=1159.915,163.524,-58.113,-178.406,6.834,148.797
C09865=1159.910,163.773,-58.135,-178.404,6.836,148.797
C09866=1159.905,164.022,-58.157,-178.400,6.838,148.796
C09867=1159.901,164.271,-58.178,-178.398,6.840,148.796
C09868=1159.896,164.520,-58.201,-178.395,6.842,148.796
C09869=1159.891,164.769,-58.222,-178.392,6.843,148.795
C09870=1159.887,165.018,-58.244,-178.390,6.846,148.795
C09871=1159.882,165.267,-58.266,-178.387,6.847,148.795
C09872=1159.878,165.516,-58.288,-178.384,6.850,148.794
C09873=1159.873,165.765,-58.310,-178.381,6.852,148.794
C09874=1159.868,166.014,-58.332,-178.379,6.853,148.794
C09875=1159.863,166.263,-58.354,-178.376,6.855,148.793
C09876=1159.858,166.512,-58.376,-178.373,6.857,148.793
C09877=1159.854,166.761,-58.398,-178.371,6.860,148.793
C09878=1159.849,167.010,-58.419,-178.368,6.861,148.792
C09879=1159.845,167.259,-58.441,-178.365,6.863,148.792
C09880=1159.839,167.508,-58.464,-178.363,6.865,148.792
C09881=1159.835,167.757,-58.486,-178.359,6.868,148.791
C09882=1159.831,168.005,-58.508,-178.357,6.869,148.791
C09883=1159.826,168.255,-58.530,-178.354,6.871,148.791
C09884=1159.822,168.504,-58.552,-178.352,6.873,148.790
C09885=1159.816,168.753,-58.575,-178.349,6.875,148.790
C09886=1159.812,169.002,-58.597,-178.346,6.877,148.790
C09887=1159.807,169.251,-58.618,-178.343,6.879,148.789
C09888=1159.803,169.500,-58.641,-178.340,6.881,148.789
C09889=1159.798,169.749,-58.663,-178.338,6.883,148.789
C09890=1159.793,169.998,-58.685,-178.335,6.886,148.788
C09891=1159.789,170.247,-58.707,-178.332,6.887,148.788
C09892=1159.784,170.496,-58.730,-178.329,6.889,148.788
C09893=1159.779,170.744,-58.752,-178.327,6.891,148.787
C09894=1159.775,170.994,-58.774,-178.324,6.893,148.787
C09895=1159.770,171.243,-58.797,-178.321,6.895,148.787
C09896=1159.765,171.491,-58.819,-178.319,6.897,148.786
C09897=1159.761,171.741,-58.841,-178.316,6.899,148.786
C09898=1159.756,171.989,-58.863,-178.313,6.901,148.786
C09899=1159.751,172.238,-58.886,-178.310,6.904,148.786
C09900=1159.747,172.488,-58.908,-178.308,6.905,148.785
C09901=1159.741,172.737,-58.931,-178.305,6.907,148.785
C09902=1159.737,172.985,-58.953,-178.302,6.909,148.784
C09903=1159.733,173.234,-58.975,-178.299,6.911,148.784
C09904=1159.728,173.483,-58.998,-178.297,6.914,148.784
C09905=1159.724,173.732,-59.020,-178.294,6.915,148.784
C09906=1159.719,173.981,-59.042,-178.291,6.917,148.783
C09907=1159.714,174.230,-59.066,-178.288,6.920,148.783
C09908=1159.710,174.479,-59.088,-178.285,6.921,148.783
C09909=1159.705,174.728,-59.111,-178.283,6.923,148.782
C09910=1159.700,174.977,-59.133,-178.280,6.926,148.782
C09911=1159.696,175.226,-59.156,-178.277,6.928,148.782
C09912=1159.691,175.475,-59.178,-178.275,6.930,148.781
C09913=1159.687,175.723,-59.200,-178.272,6.931,148.781
C09914=1159.682,175.973,-59.223,-178.269,6.934,148.781
C09915=1159.677,176.221,-59.245,-178.266,6.936,148.780
C09916=1159.672,176.471,-59.268,-178.264,6.938,148.780
C09917=1159.668,176.719,-59.291,-178.261,6.939,148.780
C09918=1159.663,176.968,-59.313,-178.258,6.942,148.780
C09919=1159.659,177.217,-59.336,-178.256,6.944,148.779
C09920=1159.654,177.466,-59.359,-178.253,6.946,148.779
C09921=1159.650,177.716,-59.381,-178.250,6.948,148.779
C09922=1159.644,177.964,-59.404,-178.247,6.951,148.778
C09923=1159.640,178.213,-59.427,-178.245,6.952,148.778
C09924=1159.635,178.462,-59.450,-178.242,6.954,148.778
C09925=1159.631,178.710,-59.472,-178.239,6.957,148.777
C09926=1159.626,178.960,-59.495,-178.237,6.959,148.777
C09927=1159.622,179.209,-59.517,-178.234,6.960,148.777
C09928=1159.617,179.458,-59.541,-178.231,6.963,148.776
C09929=1159.612,179.706,-59.564,-178.228,6.965,148.776
C09930=1159.608,179.955,-59.586,-178.226,6.967,148.776
C09931=1159.603,180.204,-59.609,-178.222,6.969,148.776
C09932=1159.599,180.453,-59.632,-178.220,6.971,148.775
C09933=1159.594,180.703,-59.655,-178.217,6.973,148.775
C09934=1159.589,180.951,-59.678,-178.215,6.975,148.775
C09935=1159.585,181.200,-59.700,-178.212,6.978,148.774
C09936=1159.580,181.449,-59.724,-178.209,6.979,148.774
C09937=1159.576,181.698,-59.747,-178.206,6.981,148.774
C09938=1159.570,181.946,-59.769,-178.203,6.984,148.774
C09939=1159.566,182.196,-59.792,-178.201,6.986,148.773
C09940=1159.562,182.444,-59.815,-178.198,6.988,148.773
C09941=1159.557,182.693,-59.838,-178.195,6.990,148.773
C09942=1159.552,182.942,-59.862,-178.193,6.992,148.772
C09943=1159.548,183.191,-59.884,-178.190,6.994,148.772
C09944=1159.543,183.440,-59.907,-178.187,6.997,148.772
C09945=1159.538,183.709,-59.932,-178.184,6.999,148.772
C09946=1159.534,183.979,-59.957,-178.181,7.001,148.771
C09947=1159.528,184.249,-59.982,-178.178,7.004,148.771
C09948=1159.523,184.519,-60.007,-178.175,7.006,148.771
C09949=1159.518,184.768,-60.031,-178.172,7.007,148.770
C09950=1159.514,185.016,-60.053,-178.170,7.010,148.770
C09951=1159.509,185.265,-60.076,-178.167,7.012,148.770
C09952=1159.504,185.514,-60.100,-178.164,7.015,148.769
C09953=1159.500,185.763,-60.123,-178.162,7.017,148.769
C09954=1159.496,186.012,-60.146,-178.159,7.018,148.769
C09955=1159.491,186.261,-60.169,-178.156,7.021,148.769
C09956=1159.486,186.510,-60.193,-178.153,7.023,148.768
C09957=1159.482,186.759,-60.216,-178.151,7.025,148.768
C09958=1159.476,187.007,-60.239,-178.147,7.027,148.768
C09959=1159.472,187.256,-60.262,-178.145,7.029,148.767
C09960=1159.468,187.505,-60.285,-178.143,7.031,148.767
C09961=1159.463,187.754,-60.308,-178.139,7.034,148.767
C09962=1159.458,188.003,-60.332,-178.137,7.036,148.766
C09963=1159.454,188.252,-60.355,-178.134,7.038,148.766
C09964=1159.449,188.501,-60.379,-178.131,7.040,148.766
C09965=1159.445,188.749,-60.403,-178.128,7.042,148.766
C09966=1159.441,188.998,-60.425,-178.126,7.045,148.766
C09967=1159.436,189.247,-60.449,-178.123,7.047,148.765
C09968=1159.431,189.496,-60.472,-178.120,7.048,148.765
C09969=1159.426,189.745,-60.495,-178.117,7.051,148.765
C09970=1159.422,189.994,-60.519,-178.115,7.053,148.764
C09971=1159.417,190.243,-60.543,-178.112,7.055,148.764
C09972=1159.413,190.492,-60.566,-178.109,7.058,148.764
C09973=1159.407,190.740,-60.589,-178.107,7.060,148.764
C09974=1159.403,190.989,-60.613,-178.104,7.062,148.763
C09975=1159.398,191.238,-60.636,-178.101,7.064,148.763
C09976=1159.394,191.487,-60.660,-178.098,7.066,148.763
C09977=1159.389,191.736,-60.683,-178.096,7.069,148.763
C09978=1159.384,191.985,-60.707,-178.093,7.071,148.762
C09979=1159.380,192.233,-60.731,-178.090,7.073,148.762
C09980=1159.375,192.482,-60.754,-178.088,7.075,148.762
C09981=1159.370,192.731,-60.778,-178.085,7.077,148.761
C09982=1159.366,192.979,-60.802,-178.082,7.080,148.761
C09983=1159.361,193.228,-60.825,-178.079,7.082,148.761
C09984=1159.357,193.478,-60.849,-178.076,7.084,148.761
C09985=1159.353,193.727,-60.873,-178.074,7.087,148.761
C09986=1159.348,193.976,-60.896,-178.071,7.088,148.760
C09987=1159.343,194.225,-60.920,-178.068,7.091,148.760
C09988=1159.339,194.473,-60.944,-178.066,7.093,148.760
C09989=1159.334,194.722,-60.967,-178.062,7.096,148.759
C09990=1159.330,194.971,-60.991,-178.060,7.097,148.759
C09991=1159.325,195.220,-61.014,-178.058,7.099,148.759
C09992=1159.321,195.468,-61.038,-178.054,7.102,148.759
C09993=1159.316,195.717,-61.062,-178.052,7.104,148.758
C09994=1159.312,195.965,-61.086,-178.049,7.107,148.758
C09995=1159.307,196.214,-61.109,-178.046,7.108,148.758
C09996=1159.302,196.464,-61.133,-178.043,7.111,148.758
//INST
///DATE 2021/06/25 14:30
///ATTR SC,RW,RJ
////FRAME ROBOT
///GROUP1 RB1
NOP
MOVL C00000 V=800.0 PL=0
MOVL C00001 V=800.0 PL=0
MOVL C00002 V=800.0 PL=0
MOVL C00003 V=800.0 PL=0
MOVL C00004 V=800.0 PL=0
MOVL C00005 V=800.0 PL=0
MOVL C00006 V=800.0 PL=0
MOVL C00007 V=800.0 PL=0
MOVL C00008 V=800.0 PL=0
MOVL C00009 V=800.0 PL=0
MOVL C00010 V=800.0 PL=0
MOVL C00011 V=800.0 PL=0
MOVL C00012 V=800.0 PL=0
MOVL C00013 V=800.0 PL=0
MOVL C00014 V=800.0 PL=0
MOVL C00015 V=800.0 PL=0
MOVL C00016 V=800.0 PL=0
MOVL C00017 V=800.0 PL=0
MOVL C00018 V=800.0 PL=0
MOVL C00019 V=800.0 PL=0
MOVL C00020 V=800.0 PL=0
MOVL C00021 V=800.0 PL=0
MOVL C00022 V=800.0 PL=0
MOVL C00023 V=800.0 PL=0
MOVL C00024 V=800.0 PL=0
MOVL C00025 V=800.0 PL=0
MOVL C00026 V=800.0 PL=0
MOVL C00027 V=800.0 PL=0
MOVL C00028 V=800.0 PL=0
MOVL C00029 V=800.0 PL=0
MOVL C00030 V=800.0 PL=0
MOVL C00031 V=800.0 PL=0
MOVL C00032 V=800.0 PL=0
MOVL C00033 V=800.0 PL=0
MOVL C00034 V=800.0 PL=0
MOVL C00035 V=800.0 PL=0
MOVL C00036 V=800.0 PL=0
MOVL C00037 V=800.0 PL=0
MOVL C00038 V=800.0 PL=0
MOVL C00039 V=800.0 PL=0
MOVL C00040 V=800.0 PL=0
MOVL C00041 V=800.0 PL=0
MOVL C00042 V=800.0 PL=0
MOVL C00043 V=800.0 PL=0
MOVL C00044 V=800.0 PL=0
MOVL C00045 V=800.0 PL=0
MOVL C00046 V=800.0 PL=0
MOVL C00047 V=800.0 PL=0
MOVL C00048 V=800.0 PL=0
MOVL C00049 V=800.0 PL=0
MOVL C00050 V=800.0 PL=0
MOVL C00051 V=800.0 PL=0
MOVL C00052 V=800.0 PL=0
MOVL C00053 V=800.0 PL=0
MOVL C00054 V=800.0 PL=0
MOVL C00055 V=800.0 PL=0
MOVL C00056 V=800.0 PL=0
MOVL C00057 V=800.0 PL=0
MOVL C00058 V=800.0 PL=0
MOVL C00059 V=800.0 PL=0
MOVL C00060 V=800.0 PL=0
MOVL C00061 V=800.0 PL=0
MOVL C00062 V=800.0 PL=0
MOVL C00063 V=800.0 PL=0
MOVL C00064 V=800.0 PL=0
MOVL C00065 V=800.0 PL=0
MOVL C00066 V=800.0 PL=0
MOVL C00067 V=800.0 PL=0
MOVL C00068 V=800.0 PL=0
MOVL C00069 V=800.0 PL=0
MOVL C00070 V=800.0 PL=0
MOVL C00071 V=800.0 PL=0
MOVL C00072 V=800.0 PL=0
MOVL C00073 V=800.0 PL=0
MOVL C00074 V=800.0 PL=0
MOVL C00075 V=800.0 PL=0
MOVL C00076 V=800.0 PL=0
MOVL C00077 V=800.0 PL=0
MOVL C00078 V=800.0 PL=0
MOVL C00079 V=800.0 PL=0
MOVL C00080 V=800.0 PL=0
MOVL C00081 V=800.0 PL=0
MOVL C00082 V=800.0 PL=0
MOVL C00083 V=800.0 PL=0
MOVL C00084 V=800.0 PL=0
MOVL C00085 V=800.0 PL=0
MOVL C00086 V=800.0 PL=0
MOVL C00087 V=800.0 PL=0
MOVL C00088 V=800.0 PL=0
MOVL C00089 V=800.0 PL=0
MOVL C00090 V=800.0 PL=0
MOVL C00091 V=800.0 PL=0
MOVL C00092 V=800.0 PL=0
MOVL C00093 V=800.0 PL=0
MOVL C00094 V=800.0 PL=0
MOVL C00095 V=800.0 PL=0
MOVL C00096 V=800.0 PL=0
MOVL C00097 V=800.0 PL=0
MOVL C00098 V=800.0 PL=0
MOVL C00099 V=800.0 PL=0
MOVL C00100 V=800.0 PL=0
MOVL C00101 V=800.0 PL=0
MOVL C00102 V=800.0 PL=0
MOVL C00103 V=800.0 PL=0
MOVL C00104 V=800.0 PL=0
MOVL C00105 V=800.0 PL=0
MOVL C00106 V=800.0 PL=0
MOVL C00107 V=800.0 PL=0
MOVL C00108 V=800.0 PL=0
MOVL C00109 V=800.0 PL=0
MOVL C00110 V=800.0 PL=0
MOVL C00111 V=800.0 PL=0
MOVL C00112 V=800.0 PL=0
MOVL C00113 V=800.0 PL=0
MOVL C00114 V=800.0 PL=0
MOVL C00115 V=800.0 PL=0
MOVL C00116 V=800.0 PL=0
MOVL C00117 V=800.0 PL=0
MOVL C00118 V=800.0 PL=0
MOVL C00119 V=800.0 PL=0
MOVL C00120 V=800.0 PL=0
MOVL C00121 V=800.0 PL=0
MOVL C00122 V=800.0 PL=0
MOVL C00123 V=800.0 PL=0
MOVL C00124 V=800.0 PL=0
MOVL C00125 V=800.0 PL=0
MOVL C00126 V=800.0 PL=0
MOVL C00127 V=800.0 PL=0
MOVL C00128 V=800.0 PL=0
MOVL C00129 V=800.0 PL=0
MOVL C00130 V=800.0 PL=0
MOVL C00131 V=800.0 PL=0
MOVL C00132 V=800.0 PL=0
MOVL C00133 V=800.0 PL=0
MOVL C00134 V=800.0 PL=0
MOVL C00135 V=800.0 PL=0
MOVL C00136 V=800.0 PL=0
MOVL C00137 V=800.0 PL=0
MOVL C00138 V=800.0 PL=0
MOVL C00139 V=800.0 PL=0
MOVL C00140 V=800.0 PL=0
MOVL C00141 V=800.0 PL=0
MOVL C00142 V=800.0 PL=0
MOVL C00143 V=800.0 PL=0
MOVL C00144 V=800.0 PL=0
MOVL C00145 V=800.0 PL=0
MOVL C00146 V=800.0 PL=0
MOVL C00147 V=800.0 PL=0
MOVL C00148 V=800.0 PL=0
MOVL C00149 V=800.0 PL=0
MOVL C00150 V=800.0 PL=0
MOVL C00151 V=800.0 PL=0
MOVL C00152 V=800.0 PL=0
MOVL C00153 V=800.0 PL=0
MOVL C00154 V=800.0 PL=0
MOVL C00155 V=800.0 PL=0
MOVL C00156 V=800.0 PL=0
MOVL C00157 V=800.0 PL=0
MOVL C00158 V=800.0 PL=0
MOVL C00159 V=800.0 PL=0
MOVL C00160 V=800.0 PL=0
MOVL C00161 V=800.0 PL=0
MOVL C00162 V=800.0 PL=0
MOVL C00163 V=800.0 PL=0
MOVL C00164 V=800.0 PL=0
MOVL C00165 V=800.0 PL=0
MOVL C00166 V=800.0 PL=0
MOVL C00167 V=800.0 PL=0
MOVL C00168 V=800.0 PL=0
MOVL C00169 V=800.0 PL=0
MOVL C00170 V=800.0 PL=0
MOVL C00171 V=800.0 PL=0
MOVL C00172 V=800.0 PL=0
MOVL C00173 V=800.0 PL=0
MOVL C00174 V=800.0 PL=0
MOVL C00175 V=800.0 PL=0
MOVL C00176 V=800.0 PL=0
MOVL C00177 V=800.0 PL=0
MOVL C00178 V=800.0 PL=0
MOVL C00179 V=800.0 PL=0
MOVL C00180 V=800.0 PL=0
MOVL C00181 V=800.0 PL=0
MOVL C00182 V=800.0 PL=0
MOVL C00183 V=800.0 PL=0
MOVL C00184 V=800.0 PL=0
MOVL C00185 V=800.0 PL=0
MOVL C00186 V=800.0 PL=0
MOVL C00187 V=800.0 PL=0
MOVL C00188 V=800.0 PL=0
MOVL C00189 V=800.0 PL=0
MOVL C00190 V=800.0 PL=0
MOVL C00191 V=800.0 PL=0
MOVL C00192 V=800.0 PL=0
MOVL C00193 V=800.0 PL=0
MOVL C00194 V=800.0 PL=0
MOVL C00195 V=800.0 PL=0
MOVL C00196 V=800.0 PL=0
MOVL C00197 V=800.0 PL=0
MOVL C00198 V=800.0 PL=0
MOVL C00199 V=800.0 PL=0
MOVL C00200 V=800.0 PL=0
MOVL C00201 V=800.0 PL=0
MOVL C00202 V=800.0 PL=0
MOVL C00203 V=800.0 PL=0
MOVL C00204 V=800.0 PL=0
MOVL C00205 V=800.0 PL=0
MOVL C00206 V=800.0 PL=0
MOVL C00207 V=800.0 PL=0
MOVL C00208 V=800.0 PL=0
MOVL C00209 V=800.0 PL=0
MOVL C00210 V=800.0 PL=0
MOVL C00211 V=800.0 PL=0
MOVL C00212 V=800.0 PL=0
MOVL C00213 V=800.0 PL=0
MOVL C00214 V=800.0 PL=0
MOVL C00215 V=800.0 PL=0
MOVL C00216 V=800.0 PL=0
MOVL C00217 V=800.0 PL=0
MOVL C00218 V=800.0 PL=0
MOVL C00219 V=800.0 PL=0
MOVL C00220 V=800.0 PL=0
MOVL C00221 V=800.0 PL=0
MOVL C00222 V=800.0 PL=0
MOVL C00223 V=800.0 PL=0
MOVL C00224 V=800.0 PL=0
MOVL C00225 V=800.0 PL=0
MOVL C00226 V=800.0 PL=0
MOVL C00227 V=800.0 PL=0
MOVL C00228 V=800.0 PL=0
MOVL C00229 V=800.0 PL=0
MOVL C00230 V=800.0 PL=0
MOVL C00231 V=800.0 PL=0
MOVL C00232 V=800.0 PL=0
MOVL C00233 V=800.0 PL=0
MOVL C00234 V=800.0 PL=0
MOVL C00235 V=800.0 PL=0
MOVL C00236 V=800.0 PL=0
MOVL C00237 V=800.0 PL=0
MOVL C00238 V=800.0 PL=0
MOVL C00239 V=800.0 PL=0
MOVL C00240 V=800.0 PL=0
MOVL C00241 V=800.0 PL=0
MOVL C00242 V=800.0 PL=0
MOVL C00243 V=800.0 PL=0
MOVL C00244 V=800.0 PL=0
MOVL C00245 V=800.0 PL=0
MOVL C00246 V=800.0 PL=0
MOVL C00247 V=800.0 PL=0
MOVL C00248 V=800.0 PL=0
MOVL C00249 V=800.0 PL=0
MOVL C00250 V=800.0 PL=0
MOVL C00251 V=800.0 PL=0
MOVL C00252 V=800.0 PL=0
MOVL C00253 V=800.0 PL=0
MOVL C00254 V=800.0 PL=0
MOVL C00255 V=800.0 PL=0
MOVL C00256 V=800.0 PL=0
MOVL C00257 V=800.0 PL=0
MOVL C00258 V=800.0 PL=0
MOVL C00259 V=800.0 PL=0
MOVL C00260 V=800.0 PL=0
MOVL C00261 V=800.0 PL=0
MOVL C00262 V=800.0 PL=0
MOVL C00263 V=800.0 PL=0
MOVL C00264 V=800.0 PL=0
MOVL C00265 V=800.0 PL=0
MOVL C00266 V=800.0 PL=0
MOVL C00267 V=800.0 PL=0
MOVL C00268 V=800.0 PL=0
MOVL C00269 V=800.0 PL=0
MOVL C00270 V=800.0 PL=0
MOVL C00271 V=800.0 PL=0
MOVL C00272 V=800.0 PL=0
MOVL C00273 V=800.0 PL=0
MOVL C00274 V=800.0 PL=0
MOVL C00275 V=800.0 PL=0
MOVL C00276 V=800.0 PL=0
MOVL C00277 V=800.0 PL=0
MOVL C00278 V=800.0 PL=0
MOVL C00279 V=800.0 PL=0
MOVL C00280 V=800.0 PL=0
MOVL C00281 V=800.0 PL=0
MOVL C00282 V=800.0 PL=0
MOVL C00283 V=800.0 PL=0
MOVL C00284 V=800.0 PL=0
MOVL C00285 V=800.0 PL=0
MOVL C00286 V=800.0 PL=0
MOVL C00287 V=800.0 PL=0
MOVL C00288 V=800.0 PL=0
MOVL C00289 V=800.0 PL=0
MOVL C00290 V=800.0 PL=0
MOVL C00291 V=800.0 PL=0
MOVL C00292 V=800.0 PL=0
MOVL C00293 V=800.0 PL=0
MOVL C00294 V=800.0 PL=0
MOVL C00295 V=800.0 PL=0
MOVL C00296 V=800.0 PL=0
MOVL C00297 V=800.0 PL=0
MOVL C00298 V=800.0 PL=0
MOVL C00299 V=800.0 PL=0
MOVL C00300 V=800.0 PL=0
MOVL C00301 V=800.0 PL=0
MOVL C00302 V=800.0 PL=0
MOVL C00303 V=800.0 PL=0
MOVL C00304 V=800.0 PL=0
MOVL C00305 V=800.0 PL=0
MOVL C00306 V=800.0 PL=0
MOVL C00307 V=800.0 PL=0
MOVL C00308 V=800.0 PL=0
MOVL C00309 V=800.0 PL=0
MOVL C00310 V=800.0 PL=0
MOVL C00311 V=800.0 PL=0
MOVL C00312 V=800.0 PL=0
MOVL C00313 V=800.0 PL=0
MOVL C00314 V=800.0 PL=0
MOVL C00315 V=800.0 PL=0
MOVL C00316 V=800.0 PL=0
MOVL C00317 V=800.0 PL=0
MOVL C00318 V=800.0 PL=0
MOVL C00319 V=800.0 PL=0
MOVL C00320 V=800.0 PL=0
MOVL C00321 V=800.0 PL=0
MOVL C00322 V=800.0 PL=0
MOVL C00323 V=800.0 PL=0
MOVL C00324 V=800.0 PL=0
MOVL C00325 V=800.0 PL=0
MOVL C00326 V=800.0 PL=0
MOVL C00327 V=800.0 PL=0
MOVL C00328 V=800.0 PL=0
MOVL C00329 V=800.0 PL=0
MOVL C00330 V=800.0 PL=0
MOVL C00331 V=800.0 PL=0
MOVL C00332 V=800.0 PL=0
MOVL C00333 V=800.0 PL=0
MOVL C00334 V=800.0 PL=0
MOVL C00335 V=800.0 PL=0
MOVL C00336 V=800.0 PL=0
MOVL C00337 V=800.0 PL=0
MOVL C00338 V=800.0 PL=0
MOVL C00339 V=800.0 PL=0
MOVL C00340 V=800.0 PL=0
MOVL C00341 V=800.0 PL=0
MOVL C00342 V=800.0 PL=0
MOVL C00343 V=800.0 PL=0
MOVL C00344 V=800.0 PL=0
MOVL C00345 V=800.0 PL=0
MOVL C00346 V=800.0 PL=0
MOVL C00347 V=800.0 PL=0
MOVL C00348 V=800.0 PL=0
MOVL C00349 V=800.0 PL=0
MOVL C00350 V=800.0 PL=0
MOVL C00351 V=800.0 PL=0
MOVL C00352 V=800.0 PL=0
MOVL C00353 V=800.0 PL=0
MOVL C00354 V=800.0 PL=0
MOVL C00355 V=800.0 PL=0
MOVL C00356 V=800.0 PL=0
MOVL C00357 V=800.0 PL=0
MOVL C00358 V=800.0 PL=0
MOVL C00359 V=800.0 PL=0
MOVL C00360 V=800.0 PL=0
MOVL C00361 V=800.0 PL=0
MOVL C00362 V=800.0 PL=0
MOVL C00363 V=800.0 PL=0
MOVL C00364 V=800.0 PL=0
MOVL C00365 V=800.0 PL=0
MOVL C00366 V=800.0 PL=0
MOVL C00367 V=800.0 PL=0
MOVL C00368 V=800.0 PL=0
MOVL C00369 V=800.0 PL=0
MOVL C00370 V=800.0 PL=0
MOVL C00371 V=800.0 PL=0
MOVL C00372 V=800.0 PL=0
MOVL C00373 V=800.0 PL=0
MOVL C00374 V=800.0 PL=0
MOVL C00375 V=800.0 PL=0
MOVL C00376 V=800.0 PL=0
MOVL C00377 V=800.0 PL=0
MOVL C00378 V=800.0 PL=0
MOVL C00379 V=800.0 PL=0
MOVL C00380 V=800.0 PL=0
MOVL C00381 V=800.0 PL=0
MOVL C00382 V=800.0 PL=0
MOVL C00383 V=800.0 PL=0
MOVL C00384 V=800.0 PL=0
MOVL C00385 V=800.0 PL=0
MOVL C00386 V=800.0 PL=0
MOVL C00387 V=800.0 PL=0
MOVL C00388 V=800.0 PL=0
MOVL C00389 V=800.0 PL=0
MOVL C00390 V=800.0 PL=0
MOVL C00391 V=800.0 PL=0
MOVL C00392 V=800.0 PL=0
MOVL C00393 V=800.0 PL=0
MOVL C00394 V=800.0 PL=0
MOVL C00395 V=800.0 PL=0
MOVL C00396 V=800.0 PL=0
MOVL C00397 V=800.0 PL=0
MOVL C00398 V=800.0 PL=0
MOVL C00399 V=800.0 PL=0
MOVL C00400 V=800.0 PL=0
MOVL C00401 V=800.0 PL=0
MOVL C00402 V=800.0 PL=0
MOVL C00403 V=800.0 PL=0
MOVL C00404 V=800.0 PL=0
MOVL C00405 V=800.0 PL=0
MOVL C00406 V=800.0 PL=0
MOVL C00407 V=800.0 PL=0
MOVL C00408 V=800.0 PL=0
MOVL C00409 V=800.0 PL=0
MOVL C00410 V=800.0 PL=0
MOVL C00411 V=800.0 PL=0
MOVL C00412 V=800.0 PL=0
MOVL C00413 V=800.0 PL=0
MOVL C00414 V=800.0 PL=0
MOVL C00415 V=800.0 PL=0
MOVL C00416 V=800.0 PL=0
MOVL C00417 V=800.0 PL=0
MOVL C00418 V=800.0 PL=0
MOVL C00419 V=800.0 PL=0
MOVL C00420 V=800.0 PL=0
MOVL C00421 V=800.0 PL=0
MOVL C00422 V=800.0 PL=0
MOVL C00423 V=800.0 PL=0
MOVL C00424 V=800.0 PL=0
MOVL C00425 V=800.0 PL=0
MOVL C00426 V=800.0 PL=0
MOVL C00427 V=800.0 PL=0
MOVL C00428 V=800.0 PL=0
MOVL C00429 V=800.0 PL=0
MOVL C00430 V=800.0 PL=0
MOVL C00431 V=800.0 PL=0
MOVL C00432 V=800.0 PL=0
MOVL C00433 V=800.0 PL=0
MOVL C00434 V=800.0 PL=0
MOVL C00435 V=800.0 PL=0
MOVL C00436 V=800.0 PL=0
MOVL C00437 V=800.0 PL=0
MOVL C00438 V=800.0 PL=0
MOVL C00439 V=800.0 PL=0
MOVL C00440 V=800.0 PL=0
MOVL C00441 V=800.0 PL=0
MOVL C00442 V=800.0 PL=0
MOVL C00443 V=800.0 PL=0
MOVL C00444 V=800.0 PL=0
MOVL C00445 V=800.0 PL=0
MOVL C00446 V=800.0 PL=0
MOVL C00447 V=800.0 PL=0
MOVL C00448 V=800.0 PL=0
MOVL C00449 V=800.0 PL=0
MOVL C00450 V=800.0 PL=0
MOVL C00451 V=800.0 PL=0
MOVL C00452 V=800.0 PL=0
MOVL C00453 V=800.0 PL=0
MOVL C00454 V=800.0 PL=0
MOVL C00455 V=800.0 PL=0
MOVL C00456 V=800.0 PL=0
MOVL C00457 V=800.0 PL=0
MOVL C00458 V=800.0 PL=0
MOVL C00459 V=800.0 PL=0
MOVL C00460 V=800.0 PL=0
MOVL C00461 V=800.0 PL=0
MOVL C00462 V=800.0 PL=0
MOVL C00463 V=800.0 PL=0
MOVL C00464 V=800.0 PL=0
MOVL C00465 V=800.0 PL=0
MOVL C00466 V=800.0 PL=0
MOVL C00467 V=800.0 PL=0
MOVL C00468 V=800.0 PL=0
MOVL C00469 V=800.0 PL=0
MOVL C00470 V=800.0 PL=0
MOVL C00471 V=800.0 PL=0
MOVL C00472 V=800.0 PL=0
MOVL C00473 V=800.0 PL=0
MOVL C00474 V=800.0 PL=0
MOVL C00475 V=800.0 PL=0
MOVL C00476 V=800.0 PL=0
MOVL C00477 V=800.0 PL=0
MOVL C00478 V=800.0 PL=0
MOVL C00479 V=800.0 PL=0
MOVL C00480 V=800.0 PL=0
MOVL C00481 V=800.0 PL=0
MOVL C00482 V=800.0 PL=0
MOVL C00483 V=800.0 PL=0
MOVL C00484 V=800.0 PL=0
MOVL C00485 V=800.0 PL=0
MOVL C00486 V=800.0 PL=0
MOVL C00487 V=800.0 PL=0
MOVL C00488 V=800.0 PL=0
MOVL C00489 V=800.0 PL=0
MOVL C00490 V=800.0 PL=0
MOVL C00491 V=800.0 PL=0
MOVL C00492 V=800.0 PL=0
MOVL C00493 V=800.0 PL=0
MOVL C00494 V=800.0 PL=0
MOVL C00495 V=800.0 PL=0
MOVL C00496 V=800.0 PL=0
MOVL C00497 V=800.0 PL=0
MOVL C00498 V=800.0 PL=0
MOVL C00499 V=800.0 PL=0
MOVL C00500 V=800.0 PL=0
MOVL C00501 V=800.0 PL=0
MOVL C00502 V=800.0 PL=0
MOVL C00503 V=800.0 PL=0
MOVL C00504 V=800.0 PL=0
MOVL C00505 V=800.0 PL=0
MOVL C00506 V=800.0 PL=0
MOVL C00507 V=800.0 PL=0
MOVL C00508 V=800.0 PL=0
MOVL C00509 V=800.0 PL=0
MOVL C00510 V=800.0 PL=0
MOVL C00511 V=800.0 PL=0
MOVL C00512 V=800.0 PL=0
MOVL C00513 V=800.0 PL=0
MOVL C00514 V=800.0 PL=0
MOVL C00515 V=800.0 PL=0
MOVL C00516 V=800.0 PL=0
MOVL C00517 V=800.0 PL=0
MOVL C00518 V=800.0 PL=0
MOVL C00519 V=800.0 PL=0
MOVL C00520 V=800.0 PL=0
MOVL C00521 V=800.0 PL=0
MOVL C00522 V=800.0 PL=0
MOVL C00523 V=800.0 PL=0
MOVL C00524 V=800.0 PL=0
MOVL C00525 V=800.0 PL=0
MOVL C00526 V=800.0 PL=0
MOVL C00527 V=800.0 PL=0
MOVL C00528 V=800.0 PL=0
MOVL C00529 V=800.0 PL=0
MOVL C00530 V=800.0 PL=0
MOVL C00531 V=800.0 PL=0
MOVL C00532 V=800.0 PL=0
MOVL C00533 V=800.0 PL=0
MOVL C00534 V=800.0 PL=0
MOVL C00535 V=800.0 PL=0
MOVL C00536 V=800.0 PL=0
MOVL C00537 V=800.0 PL=0
MOVL C00538 V=800.0 PL=0
MOVL C00539 V=800.0 PL=0
MOVL C00540 V=800.0 PL=0
MOVL C00541 V=800.0 PL=0
MOVL C00542 V=800.0 PL=0
MOVL C00543 V=800.0 PL=0
MOVL C00544 V=800.0 PL=0
MOVL C00545 V=800.0 PL=0
MOVL C00546 V=800.0 PL=0
MOVL C00547 V=800.0 PL=0
MOVL C00548 V=800.0 PL=0
MOVL C00549 V=800.0 PL=0
MOVL C00550 V=800.0 PL=0
MOVL C00551 V=800.0 PL=0
MOVL C00552 V=800.0 PL=0
MOVL C00553 V=800.0 PL=0
MOVL C00554 V=800.0 PL=0
MOVL C00555 V=800.0 PL=0
MOVL C00556 V=800.0 PL=0
MOVL C00557 V=800.0 PL=0
MOVL C00558 V=800.0 PL=0
MOVL C00559 V=800.0 PL=0
MOVL C00560 V=800.0 PL=0
MOVL C00561 V=800.0 PL=0
MOVL C00562 V=800.0 PL=0
MOVL C00563 V=800.0 PL=0
MOVL C00564 V=800.0 PL=0
MOVL C00565 V=800.0 PL=0
MOVL C00566 V=800.0 PL=0
MOVL C00567 V=800.0 PL=0
MOVL C00568 V=800.0 PL=0
MOVL C00569 V=800.0 PL=0
MOVL C00570 V=800.0 PL=0
MOVL C00571 V=800.0 PL=0
MOVL C00572 V=800.0 PL=0
MOVL C00573 V=800.0 PL=0
MOVL C00574 V=800.0 PL=0
MOVL C00575 V=800.0 PL=0
MOVL C00576 V=800.0 PL=0
MOVL C00577 V=800.0 PL=0
MOVL C00578 V=800.0 PL=0
MOVL C00579 V=800.0 PL=0
MOVL C00580 V=800.0 PL=0
MOVL C00581 V=800.0 PL=0
MOVL C00582 V=800.0 PL=0
MOVL C00583 V=800.0 PL=0
MOVL C00584 V=800.0 PL=0
MOVL C00585 V=800.0 PL=0
MOVL C00586 V=800.0 PL=0
MOVL C00587 V=800.0 PL=0
MOVL C00588 V=800.0 PL=0
MOVL C00589 V=800.0 PL=0
MOVL C00590 V=800.0 PL=0
MOVL C00591 V=800.0 PL=0
MOVL C00592 V=800.0 PL=0
MOVL C00593 V=800.0 PL=0
MOVL C00594 V=800.0 PL=0
MOVL C00595 V=800.0 PL=0
MOVL C00596 V=800.0 PL=0
MOVL C00597 V=800.0 PL=0
MOVL C00598 V=800.0 PL=0
MOVL C00599 V=800.0 PL=0
MOVL C00600 V=800.0 PL=0
MOVL C00601 V=800.0 PL=0
MOVL C00602 V=800.0 PL=0
MOVL C00603 V=800.0 PL=0
MOVL C00604 V=800.0 PL=0
MOVL C00605 V=800.0 PL=0
MOVL C00606 V=800.0 PL=0
MOVL C00607 V=800.0 PL=0
MOVL C00608 V=800.0 PL=0
MOVL C00609 V=800.0 PL=0
MOVL C00610 V=800.0 PL=0
MOVL C00611 V=800.0 PL=0
MOVL C00612 V=800.0 PL=0
MOVL C00613 V=800.0 PL=0
MOVL C00614 V=800.0 PL=0
MOVL C00615 V=800.0 PL=0
MOVL C00616 V=800.0 PL=0
MOVL C00617 V=800.0 PL=0
MOVL C00618 V=800.0 PL=0
MOVL C00619 V=800.0 PL=0
MOVL C00620 V=800.0 PL=0
MOVL C00621 V=800.0 PL=0
MOVL C00622 V=800.0 PL=0
MOVL C00623 V=800.0 PL=0
MOVL C00624 V=800.0 PL=0
MOVL C00625 V=800.0 PL=0
MOVL C00626 V=800.0 PL=0
MOVL C00627 V=800.0 PL=0
MOVL C00628 V=800.0 PL=0
MOVL C00629 V=800.0 PL=0
MOVL C00630 V=800.0 PL=0
MOVL C00631 V=800.0 PL=0
MOVL C00632 V=800.0 PL=0
MOVL C00633 V=800.0 PL=0
MOVL C00634 V=800.0 PL=0
MOVL C00635 V=800.0 PL=0
MOVL C00636 V=800.0 PL=0
MOVL C00637 V=800.0 PL=0
MOVL C00638 V=800.0 PL=0
MOVL C00639 V=800.0 PL=0
MOVL C00640 V=800.0 PL=0
MOVL C00641 V=800.0 PL=0
MOVL C00642 V=800.0 PL=0
MOVL C00643 V=800.0 PL=0
MOVL C00644 V=800.0 PL=0
MOVL C00645 V=800.0 PL=0
MOVL C00646 V=800.0 PL=0
MOVL C00647 V=800.0 PL=0
MOVL C00648 V=800.0 PL=0
MOVL C00649 V=800.0 PL=0
MOVL C00650 V=800.0 PL=0
MOVL C00651 V=800.0 PL=0
MOVL C00652 V=800.0 PL=0
MOVL C00653 V=800.0 PL=0
MOVL C00654 V=800.0 PL=0
MOVL C00655 V=800.0 PL=0
MOVL C00656 V=800.0 PL=0
MOVL C00657 V=800.0 PL=0
MOVL C00658 V=800.0 PL=0
MOVL C00659 V=800.0 PL=0
MOVL C00660 V=800.0 PL=0
MOVL C00661 V=800.0 PL=0
MOVL C00662 V=800.0 PL=0
MOVL C00663 V=800.0 PL=0
MOVL C00664 V=800.0 PL=0
MOVL C00665 V=800.0 PL=0
MOVL C00666 V=800.0 PL=0
MOVL C00667 V=800.0 PL=0
MOVL C00668 V=800.0 PL=0
MOVL C00669 V=800.0 PL=0
MOVL C00670 V=800.0 PL=0
MOVL C00671 V=800.0 PL=0
MOVL C00672 V=800.0 PL=0
MOVL C00673 V=800.0 PL=0
MOVL C00674 V=800.0 PL=0
MOVL C00675 V=800.0 PL=0
MOVL C00676 V=800.0 PL=0
MOVL C00677 V=800.0 PL=0
MOVL C00678 V=800.0 PL=0
MOVL C00679 V=800.0 PL=0
MOVL C00680 V=800.0 PL=0
MOVL C00681 V=800.0 PL=0
MOVL C00682 V=800.0 PL=0
MOVL C00683 V=800.0 PL=0
MOVL C00684 V=800.0 PL=0
MOVL C00685 V=800.0 PL=0
MOVL C00686 V=800.0 PL=0
MOVL C00687 V=800.0 PL=0
MOVL C00688 V=800.0 PL=0
MOVL C00689 V=800.0 PL=0
MOVL C00690 V=800.0 PL=0
MOVL C00691 V=800.0 PL=0
MOVL C00692 V=800.0 PL=0
MOVL C00693 V=800.0 PL=0
MOVL C00694 V=800.0 PL=0
MOVL C00695 V=800.0 PL=0
MOVL C00696 V=800.0 PL=0
MOVL C00697 V=800.0 PL=0
MOVL C00698 V=800.0 PL=0
MOVL C00699 V=800.0 PL=0
MOVL C00700 V=800.0 PL=0
MOVL C00701 V=800.0 PL=0
MOVL C00702 V=800.0 PL=0
MOVL C00703 V=800.0 PL=0
MOVL C00704 V=800.0 PL=0
MOVL C00705 V=800.0 PL=0
MOVL C00706 V=800.0 PL=0
MOVL C00707 V=800.0 PL=0
MOVL C00708 V=800.0 PL=0
MOVL C00709 V=800.0 PL=0
MOVL C00710 V=800.0 PL=0
MOVL C00711 V=800.0 PL=0
MOVL C00712 V=800.0 PL=0
MOVL C00713 V=800.0 PL=0
MOVL C00714 V=800.0 PL=0
MOVL C00715 V=800.0 PL=0
MOVL C00716 V=800.0 PL=0
MOVL C00717 V=800.0 PL=0
MOVL C00718 V=800.0 PL=0
MOVL C00719 V=800.0 PL=0
MOVL C00720 V=800.0 PL=0
MOVL C00721 V=800.0 PL=0
MOVL C00722 V=800.0 PL=0
MOVL C00723 V=800.0 PL=0
MOVL C00724 V=800.0 PL=0
MOVL C00725 V=800.0 PL=0
MOVL C00726 V=800.0 PL=0
MOVL C00727 V=800.0 PL=0
MOVL C00728 V=800.0 PL=0
MOVL C00729 V=800.0 PL=0
MOVL C00730 V=800.0 PL=0
MOVL C00731 V=800.0 PL=0
MOVL C00732 V=800.0 PL=0
MOVL C00733 V=800.0 PL=0
MOVL C00734 V=800.0 PL=0
MOVL C00735 V=800.0 PL=0
MOVL C00736 V=800.0 PL=0
MOVL C00737 V=800.0 PL=0
MOVL C00738 V=800.0 PL=0
MOVL C00739 V=800.0 PL=0
MOVL C00740 V=800.0 PL=0
MOVL C00741 V=800.0 PL=0
MOVL C00742 V=800.0 PL=0
MOVL C00743 V=800.0 PL=0
MOVL C00744 V=800.0 PL=0
MOVL C00745 V=800.0 PL=0
MOVL C00746 V=800.0 PL=0
MOVL C00747 V=800.0 PL=0
MOVL C00748 V=800.0 PL=0
MOVL C00749 V=800.0 PL=0
MOVL C00750 V=800.0 PL=0
MOVL C00751 V=800.0 PL=0
MOVL C00752 V=800.0 PL=0
MOVL C00753 V=800.0 PL=0
MOVL C00754 V=800.0 PL=0
MOVL C00755 V=800.0 PL=0
MOVL C00756 V=800.0 PL=0
MOVL C00757 V=800.0 PL=0
MOVL C00758 V=800.0 PL=0
MOVL C00759 V=800.0 PL=0
MOVL C00760 V=800.0 PL=0
MOVL C00761 V=800.0 PL=0
MOVL C00762 V=800.0 PL=0
MOVL C00763 V=800.0 PL=0
MOVL C00764 V=800.0 PL=0
MOVL C00765 V=800.0 PL=0
MOVL C00766 V=800.0 PL=0
MOVL C00767 V=800.0 PL=0
MOVL C00768 V=800.0 PL=0
MOVL C00769 V=800.0 PL=0
MOVL C00770 V=800.0 PL=0
MOVL C00771 V=800.0 PL=0
MOVL C00772 V=800.0 PL=0
MOVL C00773 V=800.0 PL=0
MOVL C00774 V=800.0 PL=0
MOVL C00775 V=800.0 PL=0
MOVL C00776 V=800.0 PL=0
MOVL C00777 V=800.0 PL=0
MOVL C00778 V=800.0 PL=0
MOVL C00779 V=800.0 PL=0
MOVL C00780 V=800.0 PL=0
MOVL C00781 V=800.0 PL=0
MOVL C00782 V=800.0 PL=0
MOVL C00783 V=800.0 PL=0
MOVL C00784 V=800.0 PL=0
MOVL C00785 V=800.0 PL=0
MOVL C00786 V=800.0 PL=0
MOVL C00787 V=800.0 PL=0
MOVL C00788 V=800.0 PL=0
MOVL C00789 V=800.0 PL=0
MOVL C00790 V=800.0 PL=0
MOVL C00791 V=800.0 PL=0
MOVL C00792 V=800.0 PL=0
MOVL C00793 V=800.0 PL=0
MOVL C00794 V=800.0 PL=0
MOVL C00795 V=800.0 PL=0
MOVL C00796 V=800.0 PL=0
MOVL C00797 V=800.0 PL=0
MOVL C00798 V=800.0 PL=0
MOVL C00799 V=800.0 PL=0
MOVL C00800 V=800.0 PL=0
MOVL C00801 V=800.0 PL=0
MOVL C00802 V=800.0 PL=0
MOVL C00803 V=800.0 PL=0
MOVL C00804 V=800.0 PL=0
MOVL C00805 V=800.0 PL=0
MOVL C00806 V=800.0 PL=0
MOVL C00807 V=800.0 PL=0
MOVL C00808 V=800.0 PL=0
MOVL C00809 V=800.0 PL=0
MOVL C00810 V=800.0 PL=0
MOVL C00811 V=800.0 PL=0
MOVL C00812 V=800.0 PL=0
MOVL C00813 V=800.0 PL=0
MOVL C00814 V=800.0 PL=0
MOVL C00815 V=800.0 PL=0
MOVL C00816 V=800.0 PL=0
MOVL C00817 V=800.0 PL=0
MOVL C00818 V=800.0 PL=0
MOVL C00819 V=800.0 PL=0
MOVL C00820 V=800.0 PL=0
MOVL C00821 V=800.0 PL=0
MOVL C00822 V=800.0 PL=0
MOVL C00823 V=800.0 PL=0
MOVL C00824 V=800.0 PL=0
MOVL C00825 V=800.0 PL=0
MOVL C00826 V=800.0 PL=0
MOVL C00827 V=800.0 PL=0
MOVL C00828 V=800.0 PL=0
MOVL C00829 V=800.0 PL=0
MOVL C00830 V=800.0 PL=0
MOVL C00831 V=800.0 PL=0
MOVL C00832 V=800.0 PL=0
MOVL C00833 V=800.0 PL=0
MOVL C00834 V=800.0 PL=0
MOVL C00835 V=800.0 PL=0
MOVL C00836 V=800.0 PL=0
MOVL C00837 V=800.0 PL=0
MOVL C00838 V=800.0 PL=0
MOVL C00839 V=800.0 PL=0
MOVL C00840 V=800.0 PL=0
MOVL C00841 V=800.0 PL=0
MOVL C00842 V=800.0 PL=0
MOVL C00843 V=800.0 PL=0
MOVL C00844 V=800.0 PL=0
MOVL C00845 V=800.0 PL=0
MOVL C00846 V=800.0 PL=0
MOVL C00847 V=800.0 PL=0
MOVL C00848 V=800.0 PL=0
MOVL C00849 V=800.0 PL=0
MOVL C00850 V=800.0 PL=0
MOVL C00851 V=800.0 PL=0
MOVL C00852 V=800.0 PL=0
MOVL C00853 V=800.0 PL=0
MOVL C00854 V=800.0 PL=0
MOVL C00855 V=800.0 PL=0
MOVL C00856 V=800.0 PL=0
MOVL C00857 V=800.0 PL=0
MOVL C00858 V=800.0 PL=0
MOVL C00859 V=800.0 PL=0
MOVL C00860 V=800.0 PL=0
MOVL C00861 V=800.0 PL=0
MOVL C00862 V=800.0 PL=0
MOVL C00863 V=800.0 PL=0
MOVL C00864 V=800.0 PL=0
MOVL C00865 V=800.0 PL=0
MOVL C00866 V=800.0 PL=0
MOVL C00867 V=800.0 PL=0
MOVL C00868 V=800.0 PL=0
MOVL C00869 V=800.0 PL=0
MOVL C00870 V=800.0 PL=0
MOVL C00871 V=800.0 PL=0
MOVL C00872 V=800.0 PL=0
MOVL C00873 V=800.0 PL=0
MOVL C00874 V=800.0 PL=0
MOVL C00875 V=800.0 PL=0
MOVL C00876 V=800.0 PL=0
MOVL C00877 V=800.0 PL=0
MOVL C00878 V=800.0 PL=0
MOVL C00879 V=800.0 PL=0
MOVL C00880 V=800.0 PL=0
MOVL C00881 V=800.0 PL=0
MOVL C00882 V=800.0 PL=0
MOVL C00883 V=800.0 PL=0
MOVL C00884 V=800.0 PL=0
MOVL C00885 V=800.0 PL=0
MOVL C00886 V=800.0 PL=0
MOVL C00887 V=800.0 PL=0
MOVL C00888 V=800.0 PL=0
MOVL C00889 V=800.0 PL=0
MOVL C00890 V=800.0 PL=0
MOVL C00891 V=800.0 PL=0
MOVL C00892 V=800.0 PL=0
MOVL C00893 V=800.0 PL=0
MOVL C00894 V=800.0 PL=0
MOVL C00895 V=800.0 PL=0
MOVL C00896 V=800.0 PL=0
MOVL C00897 V=800.0 PL=0
MOVL C00898 V=800.0 PL=0
MOVL C00899 V=800.0 PL=0
MOVL C00900 V=800.0 PL=0
MOVL C00901 V=800.0 PL=0
MOVL C00902 V=800.0 PL=0
MOVL C00903 V=800.0 PL=0
MOVL C00904 V=800.0 PL=0
MOVL C00905 V=800.0 PL=0
MOVL C00906 V=800.0 PL=0
MOVL C00907 V=800.0 PL=0
MOVL C00908 V=800.0 PL=0
MOVL C00909 V=800.0 PL=0
MOVL C00910 V=800.0 PL=0
MOVL C00911 V=800.0 PL=0
MOVL C00912 V=800.0 PL=0
MOVL C00913 V=800.0 PL=0
MOVL C00914 V=800.0 PL=0
MOVL C00915 V=800.0 PL=0
MOVL C00916 V=800.0 PL=0
MOVL C00917 V=800.0 PL=0
MOVL C00918 V=800.0 PL=0
MOVL C00919 V=800.0 PL=0
MOVL C00920 V=800.0 PL=0
MOVL C00921 V=800.0 PL=0
MOVL C00922 V=800.0 PL=0
MOVL C00923 V=800.0 PL=0
MOVL C00924 V=800.0 PL=0
MOVL C00925 V=800.0 PL=0
MOVL C00926 V=800.0 PL=0
MOVL C00927 V=800.0 PL=0
MOVL C00928 V=800.0 PL=0
MOVL C00929 V=800.0 PL=0
MOVL C00930 V=800.0 PL=0
MOVL C00931 V=800.0 PL=0
MOVL C00932 V=800.0 PL=0
MOVL C00933 V=800.0 PL=0
MOVL C00934 V=800.0 PL=0
MOVL C00935 V=800.0 PL=0
MOVL C00936 V=800.0 PL=0
MOVL C00937 V=800.0 PL=0
MOVL C00938 V=800.0 PL=0
MOVL C00939 V=800.0 PL=0
MOVL C00940 V=800.0 PL=0
MOVL C00941 V=800.0 PL=0
MOVL C00942 V=800.0 PL=0
MOVL C00943 V=800.0 PL=0
MOVL C00944 V=800.0 PL=0
MOVL C00945 V=800.0 PL=0
MOVL C00946 V=800.0 PL=0
MOVL C00947 V=800.0 PL=0
MOVL C00948 V=800.0 PL=0
MOVL C00949 V=800.0 PL=0
MOVL C00950 V=800.0 PL=0
MOVL C00951 V=800.0 PL=0
MOVL C00952 V=800.0 PL=0
MOVL C00953 V=800.0 PL=0
MOVL C00954 V=800.0 PL=0
MOVL C00955 V=800.0 PL=0
MOVL C00956 V=800.0 PL=0
MOVL C00957 V=800.0 PL=0
MOVL C00958 V=800.0 PL=0
MOVL C00959 V=800.0 PL=0
MOVL C00960 V=800.0 PL=0
MOVL C00961 V=800.0 PL=0
MOVL C00962 V=800.0 PL=0
MOVL C00963 V=800.0 PL=0
MOVL C00964 V=800.0 PL=0
MOVL C00965 V=800.0 PL=0
MOVL C00966 V=800.0 PL=0
MOVL C00967 V=800.0 PL=0
MOVL C00968 V=800.0 PL=0
MOVL C00969 V=800.0 PL=0
MOVL C00970 V=800.0 PL=0
MOVL C00971 V=800.0 PL=0
MOVL C00972 V=800.0 PL=0
MOVL C00973 V=800.0 PL=0
MOVL C00974 V=800.0 PL=0
MOVL C00975 V=800.0 PL=0
MOVL C00976 V=800.0 PL=0
MOVL C00977 V=800.0 PL=0
MOVL C00978 V=800.0 PL=0
MOVL C00979 V=800.0 PL=0
MOVL C00980 V=800.0 PL=0
MOVL C00981 V=800.0 PL=0
MOVL C00982 V=800.0 PL=0
MOVL C00983 V=800.0 PL=0
MOVL C00984 V=800.0 PL=0
MOVL C00985 V=800.0 PL=0
MOVL C00986 V=800.0 PL=0
MOVL C00987 V=800.0 PL=0
MOVL C00988 V=800.0 PL=0
MOVL C00989 V=800.0 PL=0
MOVL C00990 V=800.0 PL=0
MOVL C00991 V=800.0 PL=0
MOVL C00992 V=800.0 PL=0
MOVL C00993 V=800.0 PL=0
MOVL C00994 V=800.0 PL=0
MOVL C00995 V=800.0 PL=0
MOVL C00996 V=800.0 PL=0
MOVL C00997 V=800.0 PL=0
MOVL C00998 V=800.0 PL=0
MOVL C00999 V=800.0 PL=0
MOVL C01000 V=800.0 PL=0
MOVL C01001 V=800.0 PL=0
MOVL C01002 V=800.0 PL=0
MOVL C01003 V=800.0 PL=0
MOVL C01004 V=800.0 PL=0
MOVL C01005 V=800.0 PL=0
MOVL C01006 V=800.0 PL=0
MOVL C01007 V=800.0 PL=0
MOVL C01008 V=800.0 PL=0
MOVL C01009 V=800.0 PL=0
MOVL C01010 V=800.0 PL=0
MOVL C01011 V=800.0 PL=0
MOVL C01012 V=800.0 PL=0
MOVL C01013 V=800.0 PL=0
MOVL C01014 V=800.0 PL=0
MOVL C01015 V=800.0 PL=0
MOVL C01016 V=800.0 PL=0
MOVL C01017 V=800.0 PL=0
MOVL C01018 V=800.0 PL=0
MOVL C01019 V=800.0 PL=0
MOVL C01020 V=800.0 PL=0
MOVL C01021 V=800.0 PL=0
MOVL C01022 V=800.0 PL=0
MOVL C01023 V=800.0 PL=0
MOVL C01024 V=800.0 PL=0
MOVL C01025 V=800.0 PL=0
MOVL C01026 V=800.0 PL=0
MOVL C01027 V=800.0 PL=0
MOVL C01028 V=800.0 PL=0
MOVL C01029 V=800.0 PL=0
MOVL C01030 V=800.0 PL=0
MOVL C01031 V=800.0 PL=0
MOVL C01032 V=800.0 PL=0
MOVL C01033 V=800.0 PL=0
MOVL C01034 V=800.0 PL=0
MOVL C01035 V=800.0 PL=0
MOVL C01036 V=800.0 PL=0
MOVL C01037 V=800.0 PL=0
MOVL C01038 V=800.0 PL=0
MOVL C01039 V=800.0 PL=0
MOVL C01040 V=800.0 PL=0
MOVL C01041 V=800.0 PL=0
MOVL C01042 V=800.0 PL=0
MOVL C01043 V=800.0 PL=0
MOVL C01044 V=800.0 PL=0
MOVL C01045 V=800.0 PL=0
MOVL C01046 V=800.0 PL=0
MOVL C01047 V=800.0 PL=0
MOVL C01048 V=800.0 PL=0
MOVL C01049 V=800.0 PL=0
MOVL C01050 V=800.0 PL=0
MOVL C01051 V=800.0 PL=0
MOVL C01052 V=800.0 PL=0
MOVL C01053 V=800.0 PL=0
MOVL C01054 V=800.0 PL=0
MOVL C01055 V=800.0 PL=0
MOVL C01056 V=800.0 PL=0
MOVL C01057 V=800.0 PL=0
MOVL C01058 V=800.0 PL=0
MOVL C01059 V=800.0 PL=0
MOVL C01060 V=800.0 PL=0
MOVL C01061 V=800.0 PL=0
MOVL C01062 V=800.0 PL=0
MOVL C01063 V=800.0 PL=0
MOVL C01064 V=800.0 PL=0
MOVL C01065 V=800.0 PL=0
MOVL C01066 V=800.0 PL=0
MOVL C01067 V=800.0 PL=0
MOVL C01068 V=800.0 PL=0
MOVL C01069 V=800.0 PL=0
MOVL C01070 V=800.0 PL=0
MOVL C01071 V=800.0 PL=0
MOVL C01072 V=800.0 PL=0
MOVL C01073 V=800.0 PL=0
MOVL C01074 V=800.0 PL=0
MOVL C01075 V=800.0 PL=0
MOVL C01076 V=800.0 PL=0
MOVL C01077 V=800.0 PL=0
MOVL C01078 V=800.0 PL=0
MOVL C01079 V=800.0 PL=0
MOVL C01080 V=800.0 PL=0
MOVL C01081 V=800.0 PL=0
MOVL C01082 V=800.0 PL=0
MOVL C01083 V=800.0 PL=0
MOVL C01084 V=800.0 PL=0
MOVL C01085 V=800.0 PL=0
MOVL C01086 V=800.0 PL=0
MOVL C01087 V=800.0 PL=0
MOVL C01088 V=800.0 PL=0
MOVL C01089 V=800.0 PL=0
MOVL C01090 V=800.0 PL=0
MOVL C01091 V=800.0 PL=0
MOVL C01092 V=800.0 PL=0
MOVL C01093 V=800.0 PL=0
MOVL C01094 V=800.0 PL=0
MOVL C01095 V=800.0 PL=0
MOVL C01096 V=800.0 PL=0
MOVL C01097 V=800.0 PL=0
MOVL C01098 V=800.0 PL=0
MOVL C01099 V=800.0 PL=0
MOVL C01100 V=800.0 PL=0
MOVL C01101 V=800.0 PL=0
MOVL C01102 V=800.0 PL=0
MOVL C01103 V=800.0 PL=0
MOVL C01104 V=800.0 PL=0
MOVL C01105 V=800.0 PL=0
MOVL C01106 V=800.0 PL=0
MOVL C01107 V=800.0 PL=0
MOVL C01108 V=800.0 PL=0
MOVL C01109 V=800.0 PL=0
MOVL C01110 V=800.0 PL=0
MOVL C01111 V=800.0 PL=0
MOVL C01112 V=800.0 PL=0
MOVL C01113 V=800.0 PL=0
MOVL C01114 V=800.0 PL=0
MOVL C01115 V=800.0 PL=0
MOVL C01116 V=800.0 PL=0
MOVL C01117 V=800.0 PL=0
MOVL C01118 V=800.0 PL=0
MOVL C01119 V=800.0 PL=0
MOVL C01120 V=800.0 PL=0
MOVL C01121 V=800.0 PL=0
MOVL C01122 V=800.0 PL=0
MOVL C01123 V=800.0 PL=0
MOVL C01124 V=800.0 PL=0
MOVL C01125 V=800.0 PL=0
MOVL C01126 V=800.0 PL=0
MOVL C01127 V=800.0 PL=0
MOVL C01128 V=800.0 PL=0
MOVL C01129 V=800.0 PL=0
MOVL C01130 V=800.0 PL=0
MOVL C01131 V=800.0 PL=0
MOVL C01132 V=800.0 PL=0
MOVL C01133 V=800.0 PL=0
MOVL C01134 V=800.0 PL=0
MOVL C01135 V=800.0 PL=0
MOVL C01136 V=800.0 PL=0
MOVL C01137 V=800.0 PL=0
MOVL C01138 V=800.0 PL=0
MOVL C01139 V=800.0 PL=0
MOVL C01140 V=800.0 PL=0
MOVL C01141 V=800.0 PL=0
MOVL C01142 V=800.0 PL=0
MOVL C01143 V=800.0 PL=0
MOVL C01144 V=800.0 PL=0
MOVL C01145 V=800.0 PL=0
MOVL C01146 V=800.0 PL=0
MOVL C01147 V=800.0 PL=0
MOVL C01148 V=800.0 PL=0
MOVL C01149 V=800.0 PL=0
MOVL C01150 V=800.0 PL=0
MOVL C01151 V=800.0 PL=0
MOVL C01152 V=800.0 PL=0
MOVL C01153 V=800.0 PL=0
MOVL C01154 V=800.0 PL=0
MOVL C01155 V=800.0 PL=0
MOVL C01156 V=800.0 PL=0
MOVL C01157 V=800.0 PL=0
MOVL C01158 V=800.0 PL=0
MOVL C01159 V=800.0 PL=0
MOVL C01160 V=800.0 PL=0
MOVL C01161 V=800.0 PL=0
MOVL C01162 V=800.0 PL=0
MOVL C01163 V=800.0 PL=0
MOVL C01164 V=800.0 PL=0
MOVL C01165 V=800.0 PL=0
MOVL C01166 V=800.0 PL=0
MOVL C01167 V=800.0 PL=0
MOVL C01168 V=800.0 PL=0
MOVL C01169 V=800.0 PL=0
MOVL C01170 V=800.0 PL=0
MOVL C01171 V=800.0 PL=0
MOVL C01172 V=800.0 PL=0
MOVL C01173 V=800.0 PL=0
MOVL C01174 V=800.0 PL=0
MOVL C01175 V=800.0 PL=0
MOVL C01176 V=800.0 PL=0
MOVL C01177 V=800.0 PL=0
MOVL C01178 V=800.0 PL=0
MOVL C01179 V=800.0 PL=0
MOVL C01180 V=800.0 PL=0
MOVL C01181 V=800.0 PL=0
MOVL C01182 V=800.0 PL=0
MOVL C01183 V=800.0 PL=0
MOVL C01184 V=800.0 PL=0
MOVL C01185 V=800.0 PL=0
MOVL C01186 V=800.0 PL=0
MOVL C01187 V=800.0 PL=0
MOVL C01188 V=800.0 PL=0
MOVL C01189 V=800.0 PL=0
MOVL C01190 V=800.0 PL=0
MOVL C01191 V=800.0 PL=0
MOVL C01192 V=800.0 PL=0
MOVL C01193 V=800.0 PL=0
MOVL C01194 V=800.0 PL=0
MOVL C01195 V=800.0 PL=0
MOVL C01196 V=800.0 PL=0
MOVL C01197 V=800.0 PL=0
MOVL C01198 V=800.0 PL=0
MOVL C01199 V=800.0 PL=0
MOVL C01200 V=800.0 PL=0
MOVL C01201 V=800.0 PL=0
MOVL C01202 V=800.0 PL=0
MOVL C01203 V=800.0 PL=0
MOVL C01204 V=800.0 PL=0
MOVL C01205 V=800.0 PL=0
MOVL C01206 V=800.0 PL=0
MOVL C01207 V=800.0 PL=0
MOVL C01208 V=800.0 PL=0
MOVL C01209 V=800.0 PL=0
MOVL C01210 V=800.0 PL=0
MOVL C01211 V=800.0 PL=0
MOVL C01212 V=800.0 PL=0
MOVL C01213 V=800.0 PL=0
MOVL C01214 V=800.0 PL=0
MOVL C01215 V=800.0 PL=0
MOVL C01216 V=800.0 PL=0
MOVL C01217 V=800.0 PL=0
MOVL C01218 V=800.0 PL=0
MOVL C01219 V=800.0 PL=0
MOVL C01220 V=800.0 PL=0
MOVL C01221 V=800.0 PL=0
MOVL C01222 V=800.0 PL=0
MOVL C01223 V=800.0 PL=0
MOVL C01224 V=800.0 PL=0
MOVL C01225 V=800.0 PL=0
MOVL C01226 V=800.0 PL=0
MOVL C01227 V=800.0 PL=0
MOVL C01228 V=800.0 PL=0
MOVL C01229 V=800.0 PL=0
MOVL C01230 V=800.0 PL=0
MOVL C01231 V=800.0 PL=0
MOVL C01232 V=800.0 PL=0
MOVL C01233 V=800.0 PL=0
MOVL C01234 V=800.0 PL=0
MOVL C01235 V=800.0 PL=0
MOVL C01236 V=800.0 PL=0
MOVL C01237 V=800.0 PL=0
MOVL C01238 V=800.0 PL=0
MOVL C01239 V=800.0 PL=0
MOVL C01240 V=800.0 PL=0
MOVL C01241 V=800.0 PL=0
MOVL C01242 V=800.0 PL=0
MOVL C01243 V=800.0 PL=0
MOVL C01244 V=800.0 PL=0
MOVL C01245 V=800.0 PL=0
MOVL C01246 V=800.0 PL=0
MOVL C01247 V=800.0 PL=0
MOVL C01248 V=800.0 PL=0
MOVL C01249 V=800.0 PL=0
MOVL C01250 V=800.0 PL=0
MOVL C01251 V=800.0 PL=0
MOVL C01252 V=800.0 PL=0
MOVL C01253 V=800.0 PL=0
MOVL C01254 V=800.0 PL=0
MOVL C01255 V=800.0 PL=0
MOVL C01256 V=800.0 PL=0
MOVL C01257 V=800.0 PL=0
MOVL C01258 V=800.0 PL=0
MOVL C01259 V=800.0 PL=0
MOVL C01260 V=800.0 PL=0
MOVL C01261 V=800.0 PL=0
MOVL C01262 V=800.0 PL=0
MOVL C01263 V=800.0 PL=0
MOVL C01264 V=800.0 PL=0
MOVL C01265 V=800.0 PL=0
MOVL C01266 V=800.0 PL=0
MOVL C01267 V=800.0 PL=0
MOVL C01268 V=800.0 PL=0
MOVL C01269 V=800.0 PL=0
MOVL C01270 V=800.0 PL=0
MOVL C01271 V=800.0 PL=0
MOVL C01272 V=800.0 PL=0
MOVL C01273 V=800.0 PL=0
MOVL C01274 V=800.0 PL=0
MOVL C01275 V=800.0 PL=0
MOVL C01276 V=800.0 PL=0
MOVL C01277 V=800.0 PL=0
MOVL C01278 V=800.0 PL=0
MOVL C01279 V=800.0 PL=0
MOVL C01280 V=800.0 PL=0
MOVL C01281 V=800.0 PL=0
MOVL C01282 V=800.0 PL=0
MOVL C01283 V=800.0 PL=0
MOVL C01284 V=800.0 PL=0
MOVL C01285 V=800.0 PL=0
MOVL C01286 V=800.0 PL=0
MOVL C01287 V=800.0 PL=0
MOVL C01288 V=800.0 PL=0
MOVL C01289 V=800.0 PL=0
MOVL C01290 V=800.0 PL=0
MOVL C01291 V=800.0 PL=0
MOVL C01292 V=800.0 PL=0
MOVL C01293 V=800.0 PL=0
MOVL C01294 V=800.0 PL=0
MOVL C01295 V=800.0 PL=0
MOVL C01296 V=800.0 PL=0
MOVL C01297 V=800.0 PL=0
MOVL C01298 V=800.0 PL=0
MOVL C01299 V=800.0 PL=0
MOVL C01300 V=800.0 PL=0
MOVL C01301 V=800.0 PL=0
MOVL C01302 V=800.0 PL=0
MOVL C01303 V=800.0 PL=0
MOVL C01304 V=800.0 PL=0
MOVL C01305 V=800.0 PL=0
MOVL C01306 V=800.0 PL=0
MOVL C01307 V=800.0 PL=0
MOVL C01308 V=800.0 PL=0
MOVL C01309 V=800.0 PL=0
MOVL C01310 V=800.0 PL=0
MOVL C01311 V=800.0 PL=0
MOVL C01312 V=800.0 PL=0
MOVL C01313 V=800.0 PL=0
MOVL C01314 V=800.0 PL=0
MOVL C01315 V=800.0 PL=0
MOVL C01316 V=800.0 PL=0
MOVL C01317 V=800.0 PL=0
MOVL C01318 V=800.0 PL=0
MOVL C01319 V=800.0 PL=0
MOVL C01320 V=800.0 PL=0
MOVL C01321 V=800.0 PL=0
MOVL C01322 V=800.0 PL=0
MOVL C01323 V=800.0 PL=0
MOVL C01324 V=800.0 PL=0
MOVL C01325 V=800.0 PL=0
MOVL C01326 V=800.0 PL=0
MOVL C01327 V=800.0 PL=0
MOVL C01328 V=800.0 PL=0
MOVL C01329 V=800.0 PL=0
MOVL C01330 V=800.0 PL=0
MOVL C01331 V=800.0 PL=0
MOVL C01332 V=800.0 PL=0
MOVL C01333 V=800.0 PL=0
MOVL C01334 V=800.0 PL=0
MOVL C01335 V=800.0 PL=0
MOVL C01336 V=800.0 PL=0
MOVL C01337 V=800.0 PL=0
MOVL C01338 V=800.0 PL=0
MOVL C01339 V=800.0 PL=0
MOVL C01340 V=800.0 PL=0
MOVL C01341 V=800.0 PL=0
MOVL C01342 V=800.0 PL=0
MOVL C01343 V=800.0 PL=0
MOVL C01344 V=800.0 PL=0
MOVL C01345 V=800.0 PL=0
MOVL C01346 V=800.0 PL=0
MOVL C01347 V=800.0 PL=0
MOVL C01348 V=800.0 PL=0
MOVL C01349 V=800.0 PL=0
MOVL C01350 V=800.0 PL=0
MOVL C01351 V=800.0 PL=0
MOVL C01352 V=800.0 PL=0
MOVL C01353 V=800.0 PL=0
MOVL C01354 V=800.0 PL=0
MOVL C01355 V=800.0 PL=0
MOVL C01356 V=800.0 PL=0
MOVL C01357 V=800.0 PL=0
MOVL C01358 V=800.0 PL=0
MOVL C01359 V=800.0 PL=0
MOVL C01360 V=800.0 PL=0
MOVL C01361 V=800.0 PL=0
MOVL C01362 V=800.0 PL=0
MOVL C01363 V=800.0 PL=0
MOVL C01364 V=800.0 PL=0
MOVL C01365 V=800.0 PL=0
MOVL C01366 V=800.0 PL=0
MOVL C01367 V=800.0 PL=0
MOVL C01368 V=800.0 PL=0
MOVL C01369 V=800.0 PL=0
MOVL C01370 V=800.0 PL=0
MOVL C01371 V=800.0 PL=0
MOVL C01372 V=800.0 PL=0
MOVL C01373 V=800.0 PL=0
MOVL C01374 V=800.0 PL=0
MOVL C01375 V=800.0 PL=0
MOVL C01376 V=800.0 PL=0
MOVL C01377 V=800.0 PL=0
MOVL C01378 V=800.0 PL=0
MOVL C01379 V=800.0 PL=0
MOVL C01380 V=800.0 PL=0
MOVL C01381 V=800.0 PL=0
MOVL C01382 V=800.0 PL=0
MOVL C01383 V=800.0 PL=0
MOVL C01384 V=800.0 PL=0
MOVL C01385 V=800.0 PL=0
MOVL C01386 V=800.0 PL=0
MOVL C01387 V=800.0 PL=0
MOVL C01388 V=800.0 PL=0
MOVL C01389 V=800.0 PL=0
MOVL C01390 V=800.0 PL=0
MOVL C01391 V=800.0 PL=0
MOVL C01392 V=800.0 PL=0
MOVL C01393 V=800.0 PL=0
MOVL C01394 V=800.0 PL=0
MOVL C01395 V=800.0 PL=0
MOVL C01396 V=800.0 PL=0
MOVL C01397 V=800.0 PL=0
MOVL C01398 V=800.0 PL=0
MOVL C01399 V=800.0 PL=0
MOVL C01400 V=800.0 PL=0
MOVL C01401 V=800.0 PL=0
MOVL C01402 V=800.0 PL=0
MOVL C01403 V=800.0 PL=0
MOVL C01404 V=800.0 PL=0
MOVL C01405 V=800.0 PL=0
MOVL C01406 V=800.0 PL=0
MOVL C01407 V=800.0 PL=0
MOVL C01408 V=800.0 PL=0
MOVL C01409 V=800.0 PL=0
MOVL C01410 V=800.0 PL=0
MOVL C01411 V=800.0 PL=0
MOVL C01412 V=800.0 PL=0
MOVL C01413 V=800.0 PL=0
MOVL C01414 V=800.0 PL=0
MOVL C01415 V=800.0 PL=0
MOVL C01416 V=800.0 PL=0
MOVL C01417 V=800.0 PL=0
MOVL C01418 V=800.0 PL=0
MOVL C01419 V=800.0 PL=0
MOVL C01420 V=800.0 PL=0
MOVL C01421 V=800.0 PL=0
MOVL C01422 V=800.0 PL=0
MOVL C01423 V=800.0 PL=0
MOVL C01424 V=800.0 PL=0
MOVL C01425 V=800.0 PL=0
MOVL C01426 V=800.0 PL=0
MOVL C01427 V=800.0 PL=0
MOVL C01428 V=800.0 PL=0
MOVL C01429 V=800.0 PL=0
MOVL C01430 V=800.0 PL=0
MOVL C01431 V=800.0 PL=0
MOVL C01432 V=800.0 PL=0
MOVL C01433 V=800.0 PL=0
MOVL C01434 V=800.0 PL=0
MOVL C01435 V=800.0 PL=0
MOVL C01436 V=800.0 PL=0
MOVL C01437 V=800.0 PL=0
MOVL C01438 V=800.0 PL=0
MOVL C01439 V=800.0 PL=0
MOVL C01440 V=800.0 PL=0
MOVL C01441 V=800.0 PL=0
MOVL C01442 V=800.0 PL=0
MOVL C01443 V=800.0 PL=0
MOVL C01444 V=800.0 PL=0
MOVL C01445 V=800.0 PL=0
MOVL C01446 V=800.0 PL=0
MOVL C01447 V=800.0 PL=0
MOVL C01448 V=800.0 PL=0
MOVL C01449 V=800.0 PL=0
MOVL C01450 V=800.0 PL=0
MOVL C01451 V=800.0 PL=0
MOVL C01452 V=800.0 PL=0
MOVL C01453 V=800.0 PL=0
MOVL C01454 V=800.0 PL=0
MOVL C01455 V=800.0 PL=0
MOVL C01456 V=800.0 PL=0
MOVL C01457 V=800.0 PL=0
MOVL C01458 V=800.0 PL=0
MOVL C01459 V=800.0 PL=0
MOVL C01460 V=800.0 PL=0
MOVL C01461 V=800.0 PL=0
MOVL C01462 V=800.0 PL=0
MOVL C01463 V=800.0 PL=0
MOVL C01464 V=800.0 PL=0
MOVL C01465 V=800.0 PL=0
MOVL C01466 V=800.0 PL=0
MOVL C01467 V=800.0 PL=0
MOVL C01468 V=800.0 PL=0
MOVL C01469 V=800.0 PL=0
MOVL C01470 V=800.0 PL=0
MOVL C01471 V=800.0 PL=0
MOVL C01472 V=800.0 PL=0
MOVL C01473 V=800.0 PL=0
MOVL C01474 V=800.0 PL=0
MOVL C01475 V=800.0 PL=0
MOVL C01476 V=800.0 PL=0
MOVL C01477 V=800.0 PL=0
MOVL C01478 V=800.0 PL=0
MOVL C01479 V=800.0 PL=0
MOVL C01480 V=800.0 PL=0
MOVL C01481 V=800.0 PL=0
MOVL C01482 V=800.0 PL=0
MOVL C01483 V=800.0 PL=0
MOVL C01484 V=800.0 PL=0
MOVL C01485 V=800.0 PL=0
MOVL C01486 V=800.0 PL=0
MOVL C01487 V=800.0 PL=0
MOVL C01488 V=800.0 PL=0
MOVL C01489 V=800.0 PL=0
MOVL C01490 V=800.0 PL=0
MOVL C01491 V=800.0 PL=0
MOVL C01492 V=800.0 PL=0
MOVL C01493 V=800.0 PL=0
MOVL C01494 V=800.0 PL=0
MOVL C01495 V=800.0 PL=0
MOVL C01496 V=800.0 PL=0
MOVL C01497 V=800.0 PL=0
MOVL C01498 V=800.0 PL=0
MOVL C01499 V=800.0 PL=0
MOVL C01500 V=800.0 PL=0
MOVL C01501 V=800.0 PL=0
MOVL C01502 V=800.0 PL=0
MOVL C01503 V=800.0 PL=0
MOVL C01504 V=800.0 PL=0
MOVL C01505 V=800.0 PL=0
MOVL C01506 V=800.0 PL=0
MOVL C01507 V=800.0 PL=0
MOVL C01508 V=800.0 PL=0
MOVL C01509 V=800.0 PL=0
MOVL C01510 V=800.0 PL=0
MOVL C01511 V=800.0 PL=0
MOVL C01512 V=800.0 PL=0
MOVL C01513 V=800.0 PL=0
MOVL C01514 V=800.0 PL=0
MOVL C01515 V=800.0 PL=0
MOVL C01516 V=800.0 PL=0
MOVL C01517 V=800.0 PL=0
MOVL C01518 V=800.0 PL=0
MOVL C01519 V=800.0 PL=0
MOVL C01520 V=800.0 PL=0
MOVL C01521 V=800.0 PL=0
MOVL C01522 V=800.0 PL=0
MOVL C01523 V=800.0 PL=0
MOVL C01524 V=800.0 PL=0
MOVL C01525 V=800.0 PL=0
MOVL C01526 V=800.0 PL=0
MOVL C01527 V=800.0 PL=0
MOVL C01528 V=800.0 PL=0
MOVL C01529 V=800.0 PL=0
MOVL C01530 V=800.0 PL=0
MOVL C01531 V=800.0 PL=0
MOVL C01532 V=800.0 PL=0
MOVL C01533 V=800.0 PL=0
MOVL C01534 V=800.0 PL=0
MOVL C01535 V=800.0 PL=0
MOVL C01536 V=800.0 PL=0
MOVL C01537 V=800.0 PL=0
MOVL C01538 V=800.0 PL=0
MOVL C01539 V=800.0 PL=0
MOVL C01540 V=800.0 PL=0
MOVL C01541 V=800.0 PL=0
MOVL C01542 V=800.0 PL=0
MOVL C01543 V=800.0 PL=0
MOVL C01544 V=800.0 PL=0
MOVL C01545 V=800.0 PL=0
MOVL C01546 V=800.0 PL=0
MOVL C01547 V=800.0 PL=0
MOVL C01548 V=800.0 PL=0
MOVL C01549 V=800.0 PL=0
MOVL C01550 V=800.0 PL=0
MOVL C01551 V=800.0 PL=0
MOVL C01552 V=800.0 PL=0
MOVL C01553 V=800.0 PL=0
MOVL C01554 V=800.0 PL=0
MOVL C01555 V=800.0 PL=0
MOVL C01556 V=800.0 PL=0
MOVL C01557 V=800.0 PL=0
MOVL C01558 V=800.0 PL=0
MOVL C01559 V=800.0 PL=0
MOVL C01560 V=800.0 PL=0
MOVL C01561 V=800.0 PL=0
MOVL C01562 V=800.0 PL=0
MOVL C01563 V=800.0 PL=0
MOVL C01564 V=800.0 PL=0
MOVL C01565 V=800.0 PL=0
MOVL C01566 V=800.0 PL=0
MOVL C01567 V=800.0 PL=0
MOVL C01568 V=800.0 PL=0
MOVL C01569 V=800.0 PL=0
MOVL C01570 V=800.0 PL=0
MOVL C01571 V=800.0 PL=0
MOVL C01572 V=800.0 PL=0
MOVL C01573 V=800.0 PL=0
MOVL C01574 V=800.0 PL=0
MOVL C01575 V=800.0 PL=0
MOVL C01576 V=800.0 PL=0
MOVL C01577 V=800.0 PL=0
MOVL C01578 V=800.0 PL=0
MOVL C01579 V=800.0 PL=0
MOVL C01580 V=800.0 PL=0
MOVL C01581 V=800.0 PL=0
MOVL C01582 V=800.0 PL=0
MOVL C01583 V=800.0 PL=0
MOVL C01584 V=800.0 PL=0
MOVL C01585 V=800.0 PL=0
MOVL C01586 V=800.0 PL=0
MOVL C01587 V=800.0 PL=0
MOVL C01588 V=800.0 PL=0
MOVL C01589 V=800.0 PL=0
MOVL C01590 V=800.0 PL=0
MOVL C01591 V=800.0 PL=0
MOVL C01592 V=800.0 PL=0
MOVL C01593 V=800.0 PL=0
MOVL C01594 V=800.0 PL=0
MOVL C01595 V=800.0 PL=0
MOVL C01596 V=800.0 PL=0
MOVL C01597 V=800.0 PL=0
MOVL C01598 V=800.0 PL=0
MOVL C01599 V=800.0 PL=0
MOVL C01600 V=800.0 PL=0
MOVL C01601 V=800.0 PL=0
MOVL C01602 V=800.0 PL=0
MOVL C01603 V=800.0 PL=0
MOVL C01604 V=800.0 PL=0
MOVL C01605 V=800.0 PL=0
MOVL C01606 V=800.0 PL=0
MOVL C01607 V=800.0 PL=0
MOVL C01608 V=800.0 PL=0
MOVL C01609 V=800.0 PL=0
MOVL C01610 V=800.0 PL=0
MOVL C01611 V=800.0 PL=0
MOVL C01612 V=800.0 PL=0
MOVL C01613 V=800.0 PL=0
MOVL C01614 V=800.0 PL=0
MOVL C01615 V=800.0 PL=0
MOVL C01616 V=800.0 PL=0
MOVL C01617 V=800.0 PL=0
MOVL C01618 V=800.0 PL=0
MOVL C01619 V=800.0 PL=0
MOVL C01620 V=800.0 PL=0
MOVL C01621 V=800.0 PL=0
MOVL C01622 V=800.0 PL=0
MOVL C01623 V=800.0 PL=0
MOVL C01624 V=800.0 PL=0
MOVL C01625 V=800.0 PL=0
MOVL C01626 V=800.0 PL=0
MOVL C01627 V=800.0 PL=0
MOVL C01628 V=800.0 PL=0
MOVL C01629 V=800.0 PL=0
MOVL C01630 V=800.0 PL=0
MOVL C01631 V=800.0 PL=0
MOVL C01632 V=800.0 PL=0
MOVL C01633 V=800.0 PL=0
MOVL C01634 V=800.0 PL=0
MOVL C01635 V=800.0 PL=0
MOVL C01636 V=800.0 PL=0
MOVL C01637 V=800.0 PL=0
MOVL C01638 V=800.0 PL=0
MOVL C01639 V=800.0 PL=0
MOVL C01640 V=800.0 PL=0
MOVL C01641 V=800.0 PL=0
MOVL C01642 V=800.0 PL=0
MOVL C01643 V=800.0 PL=0
MOVL C01644 V=800.0 PL=0
MOVL C01645 V=800.0 PL=0
MOVL C01646 V=800.0 PL=0
MOVL C01647 V=800.0 PL=0
MOVL C01648 V=800.0 PL=0
MOVL C01649 V=800.0 PL=0
MOVL C01650 V=800.0 PL=0
MOVL C01651 V=800.0 PL=0
MOVL C01652 V=800.0 PL=0
MOVL C01653 V=800.0 PL=0
MOVL C01654 V=800.0 PL=0
MOVL C01655 V=800.0 PL=0
MOVL C01656 V=800.0 PL=0
MOVL C01657 V=800.0 PL=0
MOVL C01658 V=800.0 PL=0
MOVL C01659 V=800.0 PL=0
MOVL C01660 V=800.0 PL=0
MOVL C01661 V=800.0 PL=0
MOVL C01662 V=800.0 PL=0
MOVL C01663 V=800.0 PL=0
MOVL C01664 V=800.0 PL=0
MOVL C01665 V=800.0 PL=0
MOVL C01666 V=800.0 PL=0
MOVL C01667 V=800.0 PL=0
MOVL C01668 V=800.0 PL=0
MOVL C01669 V=800.0 PL=0
MOVL C01670 V=800.0 PL=0
MOVL C01671 V=800.0 PL=0
MOVL C01672 V=800.0 PL=0
MOVL C01673 V=800.0 PL=0
MOVL C01674 V=800.0 PL=0
MOVL C01675 V=800.0 PL=0
MOVL C01676 V=800.0 PL=0
MOVL C01677 V=800.0 PL=0
MOVL C01678 V=800.0 PL=0
MOVL C01679 V=800.0 PL=0
MOVL C01680 V=800.0 PL=0
MOVL C01681 V=800.0 PL=0
MOVL C01682 V=800.0 PL=0
MOVL C01683 V=800.0 PL=0
MOVL C01684 V=800.0 PL=0
MOVL C01685 V=800.0 PL=0
MOVL C01686 V=800.0 PL=0
MOVL C01687 V=800.0 PL=0
MOVL C01688 V=800.0 PL=0
MOVL C01689 V=800.0 PL=0
MOVL C01690 V=800.0 PL=0
MOVL C01691 V=800.0 PL=0
MOVL C01692 V=800.0 PL=0
MOVL C01693 V=800.0 PL=0
MOVL C01694 V=800.0 PL=0
MOVL C01695 V=800.0 PL=0
MOVL C01696 V=800.0 PL=0
MOVL C01697 V=800.0 PL=0
MOVL C01698 V=800.0 PL=0
MOVL C01699 V=800.0 PL=0
MOVL C01700 V=800.0 PL=0
MOVL C01701 V=800.0 PL=0
MOVL C01702 V=800.0 PL=0
MOVL C01703 V=800.0 PL=0
MOVL C01704 V=800.0 PL=0
MOVL C01705 V=800.0 PL=0
MOVL C01706 V=800.0 PL=0
MOVL C01707 V=800.0 PL=0
MOVL C01708 V=800.0 PL=0
MOVL C01709 V=800.0 PL=0
MOVL C01710 V=800.0 PL=0
MOVL C01711 V=800.0 PL=0
MOVL C01712 V=800.0 PL=0
MOVL C01713 V=800.0 PL=0
MOVL C01714 V=800.0 PL=0
MOVL C01715 V=800.0 PL=0
MOVL C01716 V=800.0 PL=0
MOVL C01717 V=800.0 PL=0
MOVL C01718 V=800.0 PL=0
MOVL C01719 V=800.0 PL=0
MOVL C01720 V=800.0 PL=0
MOVL C01721 V=800.0 PL=0
MOVL C01722 V=800.0 PL=0
MOVL C01723 V=800.0 PL=0
MOVL C01724 V=800.0 PL=0
MOVL C01725 V=800.0 PL=0
MOVL C01726 V=800.0 PL=0
MOVL C01727 V=800.0 PL=0
MOVL C01728 V=800.0 PL=0
MOVL C01729 V=800.0 PL=0
MOVL C01730 V=800.0 PL=0
MOVL C01731 V=800.0 PL=0
MOVL C01732 V=800.0 PL=0
MOVL C01733 V=800.0 PL=0
MOVL C01734 V=800.0 PL=0
MOVL C01735 V=800.0 PL=0
MOVL C01736 V=800.0 PL=0
MOVL C01737 V=800.0 PL=0
MOVL C01738 V=800.0 PL=0
MOVL C01739 V=800.0 PL=0
MOVL C01740 V=800.0 PL=0
MOVL C01741 V=800.0 PL=0
MOVL C01742 V=800.0 PL=0
MOVL C01743 V=800.0 PL=0
MOVL C01744 V=800.0 PL=0
MOVL C01745 V=800.0 PL=0
MOVL C01746 V=800.0 PL=0
MOVL C01747 V=800.0 PL=0
MOVL C01748 V=800.0 PL=0
MOVL C01749 V=800.0 PL=0
MOVL C01750 V=800.0 PL=0
MOVL C01751 V=800.0 PL=0
MOVL C01752 V=800.0 PL=0
MOVL C01753 V=800.0 PL=0
MOVL C01754 V=800.0 PL=0
MOVL C01755 V=800.0 PL=0
MOVL C01756 V=800.0 PL=0
MOVL C01757 V=800.0 PL=0
MOVL C01758 V=800.0 PL=0
MOVL C01759 V=800.0 PL=0
MOVL C01760 V=800.0 PL=0
MOVL C01761 V=800.0 PL=0
MOVL C01762 V=800.0 PL=0
MOVL C01763 V=800.0 PL=0
MOVL C01764 V=800.0 PL=0
MOVL C01765 V=800.0 PL=0
MOVL C01766 V=800.0 PL=0
MOVL C01767 V=800.0 PL=0
MOVL C01768 V=800.0 PL=0
MOVL C01769 V=800.0 PL=0
MOVL C01770 V=800.0 PL=0
MOVL C01771 V=800.0 PL=0
MOVL C01772 V=800.0 PL=0
MOVL C01773 V=800.0 PL=0
MOVL C01774 V=800.0 PL=0
MOVL C01775 V=800.0 PL=0
MOVL C01776 V=800.0 PL=0
MOVL C01777 V=800.0 PL=0
MOVL C01778 V=800.0 PL=0
MOVL C01779 V=800.0 PL=0
MOVL C01780 V=800.0 PL=0
MOVL C01781 V=800.0 PL=0
MOVL C01782 V=800.0 PL=0
MOVL C01783 V=800.0 PL=0
MOVL C01784 V=800.0 PL=0
MOVL C01785 V=800.0 PL=0
MOVL C01786 V=800.0 PL=0
MOVL C01787 V=800.0 PL=0
MOVL C01788 V=800.0 PL=0
MOVL C01789 V=800.0 PL=0
MOVL C01790 V=800.0 PL=0
MOVL C01791 V=800.0 PL=0
MOVL C01792 V=800.0 PL=0
MOVL C01793 V=800.0 PL=0
MOVL C01794 V=800.0 PL=0
MOVL C01795 V=800.0 PL=0
MOVL C01796 V=800.0 PL=0
MOVL C01797 V=800.0 PL=0
MOVL C01798 V=800.0 PL=0
MOVL C01799 V=800.0 PL=0
MOVL C01800 V=800.0 PL=0
MOVL C01801 V=800.0 PL=0
MOVL C01802 V=800.0 PL=0
MOVL C01803 V=800.0 PL=0
MOVL C01804 V=800.0 PL=0
MOVL C01805 V=800.0 PL=0
MOVL C01806 V=800.0 PL=0
MOVL C01807 V=800.0 PL=0
MOVL C01808 V=800.0 PL=0
MOVL C01809 V=800.0 PL=0
MOVL C01810 V=800.0 PL=0
MOVL C01811 V=800.0 PL=0
MOVL C01812 V=800.0 PL=0
MOVL C01813 V=800.0 PL=0
MOVL C01814 V=800.0 PL=0
MOVL C01815 V=800.0 PL=0
MOVL C01816 V=800.0 PL=0
MOVL C01817 V=800.0 PL=0
MOVL C01818 V=800.0 PL=0
MOVL C01819 V=800.0 PL=0
MOVL C01820 V=800.0 PL=0
MOVL C01821 V=800.0 PL=0
MOVL C01822 V=800.0 PL=0
MOVL C01823 V=800.0 PL=0
MOVL C01824 V=800.0 PL=0
MOVL C01825 V=800.0 PL=0
MOVL C01826 V=800.0 PL=0
MOVL C01827 V=800.0 PL=0
MOVL C01828 V=800.0 PL=0
MOVL C01829 V=800.0 PL=0
MOVL C01830 V=800.0 PL=0
MOVL C01831 V=800.0 PL=0
MOVL C01832 V=800.0 PL=0
MOVL C01833 V=800.0 PL=0
MOVL C01834 V=800.0 PL=0
MOVL C01835 V=800.0 PL=0
MOVL C01836 V=800.0 PL=0
MOVL C01837 V=800.0 PL=0
MOVL C01838 V=800.0 PL=0
MOVL C01839 V=800.0 PL=0
MOVL C01840 V=800.0 PL=0
MOVL C01841 V=800.0 PL=0
MOVL C01842 V=800.0 PL=0
MOVL C01843 V=800.0 PL=0
MOVL C01844 V=800.0 PL=0
MOVL C01845 V=800.0 PL=0
MOVL C01846 V=800.0 PL=0
MOVL C01847 V=800.0 PL=0
MOVL C01848 V=800.0 PL=0
MOVL C01849 V=800.0 PL=0
MOVL C01850 V=800.0 PL=0
MOVL C01851 V=800.0 PL=0
MOVL C01852 V=800.0 PL=0
MOVL C01853 V=800.0 PL=0
MOVL C01854 V=800.0 PL=0
MOVL C01855 V=800.0 PL=0
MOVL C01856 V=800.0 PL=0
MOVL C01857 V=800.0 PL=0
MOVL C01858 V=800.0 PL=0
MOVL C01859 V=800.0 PL=0
MOVL C01860 V=800.0 PL=0
MOVL C01861 V=800.0 PL=0
MOVL C01862 V=800.0 PL=0
MOVL C01863 V=800.0 PL=0
MOVL C01864 V=800.0 PL=0
MOVL C01865 V=800.0 PL=0
MOVL C01866 V=800.0 PL=0
MOVL C01867 V=800.0 PL=0
MOVL C01868 V=800.0 PL=0
MOVL C01869 V=800.0 PL=0
MOVL C01870 V=800.0 PL=0
MOVL C01871 V=800.0 PL=0
MOVL C01872 V=800.0 PL=0
MOVL C01873 V=800.0 PL=0
MOVL C01874 V=800.0 PL=0
MOVL C01875 V=800.0 PL=0
MOVL C01876 V=800.0 PL=0
MOVL C01877 V=800.0 PL=0
MOVL C01878 V=800.0 PL=0
MOVL C01879 V=800.0 PL=0
MOVL C01880 V=800.0 PL=0
MOVL C01881 V=800.0 PL=0
MOVL C01882 V=800.0 PL=0
MOVL C01883 V=800.0 PL=0
MOVL C01884 V=800.0 PL=0
MOVL C01885 V=800.0 PL=0
MOVL C01886 V=800.0 PL=0
MOVL C01887 V=800.0 PL=0
MOVL C01888 V=800.0 PL=0
MOVL C01889 V=800.0 PL=0
MOVL C01890 V=800.0 PL=0
MOVL C01891 V=800.0 PL=0
MOVL C01892 V=800.0 PL=0
MOVL C01893 V=800.0 PL=0
MOVL C01894 V=800.0 PL=0
MOVL C01895 V=800.0 PL=0
MOVL C01896 V=800.0 PL=0
MOVL C01897 V=800.0 PL=0
MOVL C01898 V=800.0 PL=0
MOVL C01899 V=800.0 PL=0
MOVL C01900 V=800.0 PL=0
MOVL C01901 V=800.0 PL=0
MOVL C01902 V=800.0 PL=0
MOVL C01903 V=800.0 PL=0
MOVL C01904 V=800.0 PL=0
MOVL C01905 V=800.0 PL=0
MOVL C01906 V=800.0 PL=0
MOVL C01907 V=800.0 PL=0
MOVL C01908 V=800.0 PL=0
MOVL C01909 V=800.0 PL=0
MOVL C01910 V=800.0 PL=0
MOVL C01911 V=800.0 PL=0
MOVL C01912 V=800.0 PL=0
MOVL C01913 V=800.0 PL=0
MOVL C01914 V=800.0 PL=0
MOVL C01915 V=800.0 PL=0
MOVL C01916 V=800.0 PL=0
MOVL C01917 V=800.0 PL=0
MOVL C01918 V=800.0 PL=0
MOVL C01919 V=800.0 PL=0
MOVL C01920 V=800.0 PL=0
MOVL C01921 V=800.0 PL=0
MOVL C01922 V=800.0 PL=0
MOVL C01923 V=800.0 PL=0
MOVL C01924 V=800.0 PL=0
MOVL C01925 V=800.0 PL=0
MOVL C01926 V=800.0 PL=0
MOVL C01927 V=800.0 PL=0
MOVL C01928 V=800.0 PL=0
MOVL C01929 V=800.0 PL=0
MOVL C01930 V=800.0 PL=0
MOVL C01931 V=800.0 PL=0
MOVL C01932 V=800.0 PL=0
MOVL C01933 V=800.0 PL=0
MOVL C01934 V=800.0 PL=0
MOVL C01935 V=800.0 PL=0
MOVL C01936 V=800.0 PL=0
MOVL C01937 V=800.0 PL=0
MOVL C01938 V=800.0 PL=0
MOVL C01939 V=800.0 PL=0
MOVL C01940 V=800.0 PL=0
MOVL C01941 V=800.0 PL=0
MOVL C01942 V=800.0 PL=0
MOVL C01943 V=800.0 PL=0
MOVL C01944 V=800.0 PL=0
MOVL C01945 V=800.0 PL=0
MOVL C01946 V=800.0 PL=0
MOVL C01947 V=800.0 PL=0
MOVL C01948 V=800.0 PL=0
MOVL C01949 V=800.0 PL=0
MOVL C01950 V=800.0 PL=0
MOVL C01951 V=800.0 PL=0
MOVL C01952 V=800.0 PL=0
MOVL C01953 V=800.0 PL=0
MOVL C01954 V=800.0 PL=0
MOVL C01955 V=800.0 PL=0
MOVL C01956 V=800.0 PL=0
MOVL C01957 V=800.0 PL=0
MOVL C01958 V=800.0 PL=0
MOVL C01959 V=800.0 PL=0
MOVL C01960 V=800.0 PL=0
MOVL C01961 V=800.0 PL=0
MOVL C01962 V=800.0 PL=0
MOVL C01963 V=800.0 PL=0
MOVL C01964 V=800.0 PL=0
MOVL C01965 V=800.0 PL=0
MOVL C01966 V=800.0 PL=0
MOVL C01967 V=800.0 PL=0
MOVL C01968 V=800.0 PL=0
MOVL C01969 V=800.0 PL=0
MOVL C01970 V=800.0 PL=0
MOVL C01971 V=800.0 PL=0
MOVL C01972 V=800.0 PL=0
MOVL C01973 V=800.0 PL=0
MOVL C01974 V=800.0 PL=0
MOVL C01975 V=800.0 PL=0
MOVL C01976 V=800.0 PL=0
MOVL C01977 V=800.0 PL=0
MOVL C01978 V=800.0 PL=0
MOVL C01979 V=800.0 PL=0
MOVL C01980 V=800.0 PL=0
MOVL C01981 V=800.0 PL=0
MOVL C01982 V=800.0 PL=0
MOVL C01983 V=800.0 PL=0
MOVL C01984 V=800.0 PL=0
MOVL C01985 V=800.0 PL=0
MOVL C01986 V=800.0 PL=0
MOVL C01987 V=800.0 PL=0
MOVL C01988 V=800.0 PL=0
MOVL C01989 V=800.0 PL=0
MOVL C01990 V=800.0 PL=0
MOVL C01991 V=800.0 PL=0
MOVL C01992 V=800.0 PL=0
MOVL C01993 V=800.0 PL=0
MOVL C01994 V=800.0 PL=0
MOVL C01995 V=800.0 PL=0
MOVL C01996 V=800.0 PL=0
MOVL C01997 V=800.0 PL=0
MOVL C01998 V=800.0 PL=0
MOVL C01999 V=800.0 PL=0
MOVL C02000 V=800.0 PL=0
MOVL C02001 V=800.0 PL=0
MOVL C02002 V=800.0 PL=0
MOVL C02003 V=800.0 PL=0
MOVL C02004 V=800.0 PL=0
MOVL C02005 V=800.0 PL=0
MOVL C02006 V=800.0 PL=0
MOVL C02007 V=800.0 PL=0
MOVL C02008 V=800.0 PL=0
MOVL C02009 V=800.0 PL=0
MOVL C02010 V=800.0 PL=0
MOVL C02011 V=800.0 PL=0
MOVL C02012 V=800.0 PL=0
MOVL C02013 V=800.0 PL=0
MOVL C02014 V=800.0 PL=0
MOVL C02015 V=800.0 PL=0
MOVL C02016 V=800.0 PL=0
MOVL C02017 V=800.0 PL=0
MOVL C02018 V=800.0 PL=0
MOVL C02019 V=800.0 PL=0
MOVL C02020 V=800.0 PL=0
MOVL C02021 V=800.0 PL=0
MOVL C02022 V=800.0 PL=0
MOVL C02023 V=800.0 PL=0
MOVL C02024 V=800.0 PL=0
MOVL C02025 V=800.0 PL=0
MOVL C02026 V=800.0 PL=0
MOVL C02027 V=800.0 PL=0
MOVL C02028 V=800.0 PL=0
MOVL C02029 V=800.0 PL=0
MOVL C02030 V=800.0 PL=0
MOVL C02031 V=800.0 PL=0
MOVL C02032 V=800.0 PL=0
MOVL C02033 V=800.0 PL=0
MOVL C02034 V=800.0 PL=0
MOVL C02035 V=800.0 PL=0
MOVL C02036 V=800.0 PL=0
MOVL C02037 V=800.0 PL=0
MOVL C02038 V=800.0 PL=0
MOVL C02039 V=800.0 PL=0
MOVL C02040 V=800.0 PL=0
MOVL C02041 V=800.0 PL=0
MOVL C02042 V=800.0 PL=0
MOVL C02043 V=800.0 PL=0
MOVL C02044 V=800.0 PL=0
MOVL C02045 V=800.0 PL=0
MOVL C02046 V=800.0 PL=0
MOVL C02047 V=800.0 PL=0
MOVL C02048 V=800.0 PL=0
MOVL C02049 V=800.0 PL=0
MOVL C02050 V=800.0 PL=0
MOVL C02051 V=800.0 PL=0
MOVL C02052 V=800.0 PL=0
MOVL C02053 V=800.0 PL=0
MOVL C02054 V=800.0 PL=0
MOVL C02055 V=800.0 PL=0
MOVL C02056 V=800.0 PL=0
MOVL C02057 V=800.0 PL=0
MOVL C02058 V=800.0 PL=0
MOVL C02059 V=800.0 PL=0
MOVL C02060 V=800.0 PL=0
MOVL C02061 V=800.0 PL=0
MOVL C02062 V=800.0 PL=0
MOVL C02063 V=800.0 PL=0
MOVL C02064 V=800.0 PL=0
MOVL C02065 V=800.0 PL=0
MOVL C02066 V=800.0 PL=0
MOVL C02067 V=800.0 PL=0
MOVL C02068 V=800.0 PL=0
MOVL C02069 V=800.0 PL=0
MOVL C02070 V=800.0 PL=0
MOVL C02071 V=800.0 PL=0
MOVL C02072 V=800.0 PL=0
MOVL C02073 V=800.0 PL=0
MOVL C02074 V=800.0 PL=0
MOVL C02075 V=800.0 PL=0
MOVL C02076 V=800.0 PL=0
MOVL C02077 V=800.0 PL=0
MOVL C02078 V=800.0 PL=0
MOVL C02079 V=800.0 PL=0
MOVL C02080 V=800.0 PL=0
MOVL C02081 V=800.0 PL=0
MOVL C02082 V=800.0 PL=0
MOVL C02083 V=800.0 PL=0
MOVL C02084 V=800.0 PL=0
MOVL C02085 V=800.0 PL=0
MOVL C02086 V=800.0 PL=0
MOVL C02087 V=800.0 PL=0
MOVL C02088 V=800.0 PL=0
MOVL C02089 V=800.0 PL=0
MOVL C02090 V=800.0 PL=0
MOVL C02091 V=800.0 PL=0
MOVL C02092 V=800.0 PL=0
MOVL C02093 V=800.0 PL=0
MOVL C02094 V=800.0 PL=0
MOVL C02095 V=800.0 PL=0
MOVL C02096 V=800.0 PL=0
MOVL C02097 V=800.0 PL=0
MOVL C02098 V=800.0 PL=0
MOVL C02099 V=800.0 PL=0
MOVL C02100 V=800.0 PL=0
MOVL C02101 V=800.0 PL=0
MOVL C02102 V=800.0 PL=0
MOVL C02103 V=800.0 PL=0
MOVL C02104 V=800.0 PL=0
MOVL C02105 V=800.0 PL=0
MOVL C02106 V=800.0 PL=0
MOVL C02107 V=800.0 PL=0
MOVL C02108 V=800.0 PL=0
MOVL C02109 V=800.0 PL=0
MOVL C02110 V=800.0 PL=0
MOVL C02111 V=800.0 PL=0
MOVL C02112 V=800.0 PL=0
MOVL C02113 V=800.0 PL=0
MOVL C02114 V=800.0 PL=0
MOVL C02115 V=800.0 PL=0
MOVL C02116 V=800.0 PL=0
MOVL C02117 V=800.0 PL=0
MOVL C02118 V=800.0 PL=0
MOVL C02119 V=800.0 PL=0
MOVL C02120 V=800.0 PL=0
MOVL C02121 V=800.0 PL=0
MOVL C02122 V=800.0 PL=0
MOVL C02123 V=800.0 PL=0
MOVL C02124 V=800.0 PL=0
MOVL C02125 V=800.0 PL=0
MOVL C02126 V=800.0 PL=0
MOVL C02127 V=800.0 PL=0
MOVL C02128 V=800.0 PL=0
MOVL C02129 V=800.0 PL=0
MOVL C02130 V=800.0 PL=0
MOVL C02131 V=800.0 PL=0
MOVL C02132 V=800.0 PL=0
MOVL C02133 V=800.0 PL=0
MOVL C02134 V=800.0 PL=0
MOVL C02135 V=800.0 PL=0
MOVL C02136 V=800.0 PL=0
MOVL C02137 V=800.0 PL=0
MOVL C02138 V=800.0 PL=0
MOVL C02139 V=800.0 PL=0
MOVL C02140 V=800.0 PL=0
MOVL C02141 V=800.0 PL=0
MOVL C02142 V=800.0 PL=0
MOVL C02143 V=800.0 PL=0
MOVL C02144 V=800.0 PL=0
MOVL C02145 V=800.0 PL=0
MOVL C02146 V=800.0 PL=0
MOVL C02147 V=800.0 PL=0
MOVL C02148 V=800.0 PL=0
MOVL C02149 V=800.0 PL=0
MOVL C02150 V=800.0 PL=0
MOVL C02151 V=800.0 PL=0
MOVL C02152 V=800.0 PL=0
MOVL C02153 V=800.0 PL=0
MOVL C02154 V=800.0 PL=0
MOVL C02155 V=800.0 PL=0
MOVL C02156 V=800.0 PL=0
MOVL C02157 V=800.0 PL=0
MOVL C02158 V=800.0 PL=0
MOVL C02159 V=800.0 PL=0
MOVL C02160 V=800.0 PL=0
MOVL C02161 V=800.0 PL=0
MOVL C02162 V=800.0 PL=0
MOVL C02163 V=800.0 PL=0
MOVL C02164 V=800.0 PL=0
MOVL C02165 V=800.0 PL=0
MOVL C02166 V=800.0 PL=0
MOVL C02167 V=800.0 PL=0
MOVL C02168 V=800.0 PL=0
MOVL C02169 V=800.0 PL=0
